// This is what lets a reporter be slow without blocking a test. Anything that

// takes time - a file write, an ADS call - is STARTED in one of the notification

// methods and ADVANCED here.
METHOD CyclicLogic
VAR
	i : DINT;
END_VAR
FOR i := 0 TO TO_DINT(_Count) - 1 DO
	_Reporters[i].CyclicLogic();
END_FOR
END_METHOD

// Never silent, and never reported as a test failure.

//

// Reaching here with nothing attached IS silent, and there is nothing this object

// can do about it. That is what ReporterCount exists for: assert it in CI.
METHOD FrameworkError
VAR_INPUT
	Source	: T_MaxString;
	Message : T_MaxString;
END_VAR

VAR
	i : DINT;
END_VAR
IF _IsSuspended THEN
	RETURN;
END_IF

FOR i := 0 TO TO_DINT(_Count) - 1 DO
	_Reporters[i].FrameworkError(Source := Source, Message := Message);
END_FOR
END_METHOD

// FALSE while ANY attached sink still has work in flight.

//

// CI must wait for this as well as IsComplete. A run finishing and its result

// document reaching disk are different events, and copying between them yields a

// truncated artifact - which reads as a broken pipeline rather than a finished

// run.

//

// TRUE with nothing attached: no sink, no pending work.
PROPERTY IsIdle : BOOL
GET
VAR
	i : DINT;
END_VAR
IsIdle := TRUE;
FOR i := 0 TO TO_DINT(_Count) - 1 DO
	IF NOT _Reporters[i].IsIdle THEN
		IsIdle := FALSE;
		RETURN;
	END_IF
END_FOR
END_GET
END_PROPERTY

// Notify sinks again. Nothing that happened while suspended is replayed - it was

// deliberately not recorded.
METHOD Resume
_IsSuspended := FALSE;
END_METHOD

METHOD RunFinished
VAR_INPUT
	Status	   : I_TestRunStatus;
	TargetInfo : T_MaxString;
END_VAR

VAR
	i : DINT;
END_VAR
IF _IsSuspended THEN
	RETURN;
END_IF

FOR i := 0 TO TO_DINT(_Count) - 1 DO
	_Reporters[i].RunFinished(Status := Status, TargetInfo := TargetInfo);
END_FOR
END_METHOD

METHOD RunStarted
VAR_INPUT
	Label	   : T_MaxString;
	TargetInfo : T_MaxString;
END_VAR

VAR
	i : DINT;
END_VAR
IF _IsSuspended THEN
	RETURN;
END_IF

FOR i := 0 TO TO_DINT(_Count) - 1 DO
	_Reporters[i].RunStarted(Label := Label, TargetInfo := TargetInfo);
END_FOR
END_METHOD

METHOD SuiteFinished
VAR_INPUT
	Status : I_TestRunStatus;
END_VAR

VAR
	i : DINT;
END_VAR
IF _IsSuspended THEN
	RETURN;
END_IF

FOR i := 0 TO TO_DINT(_Count) - 1 DO
	_Reporters[i].SuiteFinished(Status);
END_FOR
END_METHOD

// Stop notifying sinks. Used for an individual re-run, which must not pollute the

// CI artifact with duplicate entries.

//

// Work already in flight is unaffected - CyclicLogic keeps running - so a document

// being written when this is called still lands.
METHOD Suspend
_IsSuspended := TRUE;
END_METHOD

METHOD TestFinished
VAR_INPUT
	SuiteLabel	  : T_MaxString;
	TestLabel	  : T_MaxString;
	Location	  : T_MaxString;
	Status		  : E_TestStatus;
	Kind		  : E_FailureKind;
	Summary		  : T_MaxString;
	ElapsedTime	  : LREAL;
	ElapsedCycles : UDINT;
	Assertions	  : UDINT;
END_VAR

VAR
	i : DINT;
END_VAR
IF _IsSuspended THEN
	RETURN;
END_IF

FOR i := 0 TO TO_DINT(_Count) - 1 DO
	_Reporters[i].TestFinished(SuiteLabel	 := SuiteLabel,
							   TestLabel	 := TestLabel,
							   Location		 := Location,
							   Status		 := Status,
							   Kind			 := Kind,
							   Summary		 := Summary,
							   ElapsedTime	 := ElapsedTime,
							   ElapsedCycles := ElapsedCycles,
							   Assertions	 := Assertions);
END_FOR
END_METHOD

// Only the sinks that asked for checks. A reporter that does not implement

// I_TestDetailSink is skipped without a query and without an empty method body.
METHOD TestStarted
VAR_INPUT
	SuiteLabel : T_MaxString;
	TestLabel  : T_MaxString;
	Location   : T_MaxString;
END_VAR

VAR
	i : DINT;
END_VAR
IF _IsSuspended THEN
	RETURN;
END_IF

FOR i := 0 TO TO_DINT(_Count) - 1 DO
	IF _DetailSinks[i] <> 0 THEN
		_DetailSinks[i].TestStarted(SuiteLabel := SuiteLabel, TestLabel := TestLabel, Location := Location);
	END_IF
END_FOR
END_METHOD

END_FUNCTION_BLOCK

// ---- POUs/TestArbiter.TcPOU
// Which test runs next, and when there are no more.

//

// Separated from the runner because it is the ordering POLICY and the runner is

// the test LIFECYCLE - two different reasons to change. Everything a sequencer

// parks for later lands here and nowhere else: stop on first failing test, retry,

// preconditions. Today it walks the set in registration order, and that is all it

// should do.

//

// Not generic, and holds nothing generic. It reaches the registered set through

// I_TestRoster, which is read-only: an object that decides what runs next has no

// business registering a test or clearing a verdict.
FUNCTION_BLOCK TestArbiter
VAR
	_Roster : I_TestRoster;

	// The active test. A null Test member means none - there is no sentinel index.
	_Current : ST_TestSlot;
	_Count	 : DINT;

	// Where the NEXT Advance will look. Not the active index: that lives on

	// _Current, which is the only place it is meaningful.
	_Next : DINT;

	// Never written. Assigned to _Current to clear it, so "nothing active" is one

	// well-defined value rather than six field assignments to keep in step.
	_EmptySlot : ST_TestSlot;
END_VAR

(*
	No cyclic body. Advance is called by the suite when the active test finishes,
	not every scan.
*)

// Stop the pass where it is. Called when Enable drops: the active test, and any

// setup or teardown in flight, are cancelled by the runner and the pass does not

// resume.

//

// The remaining tests are NOT visited. A run that was abandoned mid-way has not

// been run, and reporting the rest as anything - passed, failed, skipped - would

// be inventing a result.
METHOD Abandon
_Current := _EmptySlot;
_Next	 := _Count;
END_METHOD

// Move to the next test. Returns TRUE when there is one, FALSE when the pass is

// over.

//

// The return value is the whole "are we finished" mechanism, so a caller cannot

// reach a test without first having been told there is one.
METHOD Advance : BOOL
Advance	 := FALSE;
_Current := _EmptySlot;
IF (_Roster = 0) OR (_Next >= _Count) THEN
	_Next := _Count;
	RETURN;
END_IF

_Current := _Roster.Slot(_Next);
_Next	 := _Next + 1;

// A slot inside the registered range always carries a test. If one does not, the

// registry and the count disagree, and running nothing is safer than dereferencing

// a null.
Advance := (_Current.Test <> 0);
END_METHOD

// Point the arbiter at the registered set. Called once by the suite at

// composition, before any run.

//

// An interface, not the registry itself: TestRegistry is generic and cannot be

// held by its concrete type here. That constraint turned out to be the thing that

// is what makes that workable - an interface reference carries no

// generic argument, so the arbiter can hold the set AND stay non-generic.
METHOD Attach
VAR_INPUT
	Roster : I_TestRoster;
END_VAR
_Roster := Roster;
END_METHOD

// Start a pass over the registered set, in registration order.

//

// Also what a re-run calls: a re-run re-executes the registered set from the

// start, so there is no separate restart path to keep in step with this one.

//

// The count is read here, once, rather than per Advance. Registration is closed by

// the time a run starts, so it cannot change underneath the pass.
METHOD Begin
_Current := _EmptySlot;
_Next	 := 0;
IF _Roster = 0 THEN
	// Nothing attached. An empty pass rather than a fault: IsExhausted goes TRUE

	// immediately and the suite completes instead of waiting for a test that will
	// never come.
	_Count := 0;
	RETURN;
END_IF

_Count := TO_DINT(_Roster.Count);
END_METHOD

// The active test, with its label, its index and its resolved hooks. Its Test

// member is NULL when nothing is active, which is the question callers ask.

//

// "None" is a null reference, not a sentinel

// index. The index is still here - a slot carries its own position, so the runner

// can reach the matching journal - but it is carried BY the thing that is null

// when there is nothing, rather than standing in for it.
PROPERTY Current : ST_TestSlot
GET
Current := _Current;
END_GET
END_PROPERTY

// TRUE while a test is active.

//

// Letting index 0 double as "no active test" is the trap here, and the note

// why that could not work is what CHAR_SerialExecution pins. Here there is no

// index to misread: the question is whether a reference is null.
PROPERTY HasCurrent : BOOL
GET
HasCurrent := (_Current.Test <> 0);
END_GET
END_PROPERTY

// Every registered test has been visited, or the pass was abandoned. What the

// suite reads to decide the run is over.

//

// Both conditions are required. After the last test is selected the pass has

// nothing left to give out, but that test is still running - reporting the suite

// complete there would cut it off.

//

// TRUE immediately for a pass over an empty set: a suite with nothing registered

// is complete, not stuck, or any sequencer aggregating it waits forever.
PROPERTY IsExhausted : BOOL
GET
IsExhausted := (_Next >= _Count) AND (_Current.Test = 0);
END_GET
END_PROPERTY

END_FUNCTION_BLOCK

// ---- POUs/TestDeadline.TcPOU
// Bounds one phase that is not the test body: setup, or teardown.

//

// The body's deadline stays in TestJournal, which already counts that phase's

// scans and already owns the verdict an expiry produces. This object exists for

// the two phases nothing else is watching.

//

// Teardown is the reason it exists at all. TestJournal.Tick returns immediately

// once the verdict is terminal, and teardown runs after the verdict by

// definition - so before this, teardown had no deadline of any kind. On a rig

// that means an axis left powered.

//

// Self-contained: its own clock and its own scan count, because setup runs before

// the body has a first cycle and teardown runs after the journal has stopped.

// Neither span is one the journal is measuring.
FUNCTION_BLOCK TestDeadline
VAR
	_Phase		   : T_MaxString;
	_Budget		   : ST_TestBudget;
	_ElapsedCycles : UDINT;
	_Stopwatch	   : TestStopwatch;
	_IsArmed	   : BOOL;
	_Diagnostic	   : T_MaxString;
END_VAR

(*
	No cyclic body. Tick is called by the runner while the phase is in progress,
	and only then.
*)

// Start bounding a phase. Restarts the clock and the scan count.

//

// The budget passed here is the RESOLVED one - the test's own, or the suite

// default it inherited. The IsSet flags have already done their work by this

// point and are not read.
METHOD Arm
VAR_INPUT
	// 'setup' or 'teardown'. Appears in the diagnostic, so a reader can tell which

	// phase hung without opening the test.
	Phase  : T_MaxString;
	Budget : ST_TestBudget;
END_VAR
_Phase		   := Phase;
_Budget		   := Budget;
_ElapsedCycles := 0;
_Diagnostic	   := '';
_IsArmed	   := TRUE;
_Stopwatch.Start();
END_METHOD

// Why it expired, in the shared wording. Empty until it does.
PROPERTY Diagnostic : T_MaxString
GET
Diagnostic := _Diagnostic;
END_GET
END_PROPERTY

// The phase finished on its own. Stops the clock and leaves any diagnostic

// already composed intact.
METHOD Disarm
_IsArmed := FALSE;
_Stopwatch.Stop();
END_METHOD

// Scans this phase has consumed.
PROPERTY ElapsedCycles : UDINT
GET
ElapsedCycles := _ElapsedCycles;
END_GET
END_PROPERTY

PROPERTY IsArmed : BOOL
GET
IsArmed := _IsArmed;
END_GET
END_PROPERTY

// Advance one scan. Returns TRUE on the scan the deadline expires, and FALSE

// every scan after that - the caller acts once.

//

// Called AFTER the phase has run, so a budget of one allows one execution. This

// matches TestJournal.Tick deliberately: two deadline mechanisms that counted

// differently would be a trap.
METHOD Tick : BOOL
Tick := FALSE;
IF NOT _IsArmed THEN
	RETURN;
END_IF

_ElapsedCycles := _ElapsedCycles + 1;
IF (_Budget.Cycles > 0) AND (_ElapsedCycles >= _Budget.Cycles) THEN
	_Diagnostic := TestTimeoutDiagnostic(Phase	  := _Phase,
										 Cycles	  := _Budget.Cycles,
										 Timeout  := _Budget.Timeout,
										 ByCycles := TRUE);

	THIS^.Disarm();
	Tick := TRUE;
	RETURN;
END_IF

IF (_Budget.Timeout > T#0S) AND (_Stopwatch.Elapsed >= (TO_LREAL(TIME_TO_UDINT(_Budget.Timeout)) / 1000.0)) THEN
	_Diagnostic := TestTimeoutDiagnostic(Phase	  := _Phase,
										 Cycles	  := _Budget.Cycles,
										 Timeout  := _Budget.Timeout,
										 ByCycles := FALSE);

	THIS^.Disarm();
	Tick := TRUE;
END_IF
END_METHOD

END_FUNCTION_BLOCK

// ---- POUs/TestEventReporter.TcPOU
// Raises TwinCAT 3 EventLogger events for test results.

//

// The sink for anything an operator or an HMI will see: structured, timestamped,

// localizable, and filterable by event class and ID - which ADSLOGSTR output is

// not. TestLogReporter remains the sink to reach for when no project setup is

// wanted.

//

// REQUIRES the TestHarnessEvents event class in the System Type System. TwinCAT

// generates TC_Events.TestHarnessEvents from it, and every event raised below is a

// member of that.

//

// Naming the generated members rather than a GUID is deliberate: if the class is

// not registered the symbol does not resolve and this FAILS TO COMPILE, which is a

// far better failure than raising events the logger has no name for.

//

// Severity comes from the class definition too, so it is declared once - one event

// ID per outcome, each carrying its own severity.

//

// It implements I_TestReporter and NOT I_TestDetailSink. An operator-facing log

// wants verdicts; an event per individual check would bury them.

//

// Severity is not decoration. A FAILURE is Error - the code was shown to be wrong.

// An ERROR is Warning - the test could not run, so nothing was shown about the

// code at all. A build should react differently to each, and so should whoever is

// looking at the Logged Events window.
FUNCTION_BLOCK TestEventReporter IMPLEMENTS I_TestReporter
VAR
	_Message	   : FB_TcMessage;
	_IncludePasses : BOOL;
	_EventsSent	   : UDINT;
	_FailedSends   : UDINT;
	_LastError	   : HRESULT;
END_VAR

(*
	No cyclic body. Everything this sink does happens inside the notification that
	prompted it.
*)

// Nothing to advance. Send hands the message to the EventLogger and returns; the

// logger owns what happens next.
METHOD CyclicLogic
(*
	Deliberately empty. This sink starts no work it has to finish, which is also
	why IsIdle is always TRUE.
*)
END_METHOD

// The one place an event is raised. Private, so the class, the severity mapping

// and the argument handling cannot drift between call sites.
METHOD Emit
VAR_INPUT
	// A member of TC_Events.TestHarnessEvents. Carries the class GUID, the ID and

	// the severity, all three declared once in the .tmc.
	EventEntry : TcEventEntry;
	Line	   : T_MaxString;
END_VAR

VAR
	Arguments : I_TcArguments;
	Result	  : HRESULT;
END_VAR
// CreateEx, not Create: it takes the whole definition, so the class, the ID and

// the severity all come from the .tmc and none of them is restated here.

//

// ipSourceInfo 0 means "generate it", which yields the symbol path of this

// instance - the reason a raised event names the test that raised it without
// being told.
Result := _Message.CreateEx(stEventEntry := EventEntry, ipSourceInfo := 0);
IF Result < 0 THEN
	_LastError	 := Result;
	_FailedSends := _FailedSends + 1;
	RETURN;
END_IF

// ipArguments is a PROPERTY returning an interface. TwinCAT will not take a member

// off the result of a call, so it goes into a variable first.
Arguments := _Message.ipArguments;
IF Arguments <> 0 THEN
	// Cleared every time: the instance is reused, and arguments left over from the
	// previous event would be appended to this one.
	Arguments.Clear();
	Arguments.AddString(Line);
END_IF

// 0 means "use the current timestamp".
Result := _Message.Send(0);
IF Result < 0 THEN
	_LastError	 := Result;
	_FailedSends := _FailedSends + 1;
	RETURN;
END_IF

_EventsSent := _EventsSent + 1;

// Release the instance the logger created. Without it, a long run leaks one per

// event - which would show up as memory growth rather than as anything obviously

// wrong with the test results.
_Message.Release();
END_METHOD

// Events accepted by the logger. Assert it in CI if events are the artifact.
PROPERTY EventsSent : UDINT
GET
EventsSent := _EventsSent;
END_GET
END_PROPERTY

// Create or Send returned a failing HRESULT.

//

// Counted rather than swallowed. A sink that cannot deliver and cannot say so is

// indistinguishable from a run that never happened.
PROPERTY FailedSends : UDINT
GET
FailedSends := _FailedSends;
END_GET
END_PROPERTY

METHOD FrameworkError
VAR_INPUT
	Source	: T_MaxString;
	Message : T_MaxString;
END_VAR
// Never silent, never suppressed by verbosity, and never reported as a test

// failure. This is the framework saying it could not do something.

//

// One ID for every framework error. The alternative was an event class growing a

// member for each new kind, which puts the class and this file permanently in step
// with each other.
THIS^.Emit(TC_Events.TestHarnessEvents.RegistrationRejected, CONCAT(CONCAT(Source, ': '), Message));
END_METHOD

// Always TRUE. Send hands the message over and returns; this sink never holds a

// run open waiting for the logger.
PROPERTY IsIdle : BOOL
GET
IsIdle := TRUE;
END_GET
END_PROPERTY

// The most recent failing HRESULT, or zero. 16#0 means nothing has gone wrong.
PROPERTY LastError : HRESULT
GET
LastError := _LastError;
END_GET
END_PROPERTY

METHOD RunFinished
VAR_INPUT
	Status	   : I_TestRunStatus;
	TargetInfo : T_MaxString;
END_VAR

VAR
	Line	: T_MaxString;
	Outcome : E_RunOutcome;
END_VAR
IF Status = 0 THEN
	RETURN;
END_IF

// TargetInfo identifies where the run happened. Without it a matrix run across

// several targets produces events that cannot be told apart.
Line := CONCAT(CONCAT(THIS^.Tally(Status), '  on '), TargetInfo);
// Read into a variable, as SuiteFinished does: TwinCAT will not take a CASE
// selector off a property call.
Outcome := Status.Outcome;
// The same four outcomes as the suite, each with its own event. RunSkipped and
// RunErrored were added to the class for this: a skipped run is not red, and an
// errored one showed nothing about the code, so neither is a RunFailed.
CASE Outcome OF
	E_RunOutcome.Passed:
		THIS^.Emit(TC_Events.TestHarnessEvents.RunPassed, Line);
	E_RunOutcome.Skipped:
		THIS^.Emit(TC_Events.TestHarnessEvents.RunSkipped, Line);
	E_RunOutcome.Errored:
		THIS^.Emit(TC_Events.TestHarnessEvents.RunErrored, Line);
ELSE
	THIS^.Emit(TC_Events.TestHarnessEvents.RunFailed, Line);
END_CASE
END_METHOD

// Deliberately raises nothing.

//

// A banner is a LOG device: it exists because log lines are an undifferentiated

// stream that a reader scrolls through. Events are already discrete, timestamped

// and filterable by class and ID, so bracketing them would add noise to a view

// that does not need it.
METHOD RunStarted
VAR_INPUT
	Label	   : T_MaxString;
	TargetInfo : T_MaxString;
END_VAR
(*
	Nothing. See the declaration.
*)
END_METHOD

// Whether passing tests raise an event of their own. Skipped tests do not: the

// event class has no per-test skipped event, so a skip is carried by the suite's

// SuiteSkipped event until the class gains one.

//

// Off by default. Eighty Info events bury the two Errors, and the counts are

// already available through I_TestRunStatus. The Verbose severity exists for this

// and is filtered out of most views anyway - but not raising them at all is

// cheaper still.
METHOD SetVerbosity
VAR_INPUT
	IncludePasses : BOOL;
END_VAR
_IncludePasses := IncludePasses;
END_METHOD

METHOD SuiteFinished
VAR_INPUT
	Status : I_TestRunStatus;
END_VAR

VAR
	Line	: T_MaxString;
	Outcome : E_RunOutcome;
END_VAR
IF Status = 0 THEN
	RETURN;
END_IF

Line := CONCAT(CONCAT(Status.Label, ': '), THIS^.Tally(Status));

// Read into a variable: a property call is a call, and TwinCAT will not take a

// CASE selector off one any more than it will take a member.
Outcome := Status.Outcome;
// A distinct event ID per outcome, so a filtered view can show suite results

// without showing every individual failure.
CASE Outcome OF
	E_RunOutcome.Passed:
		THIS^.Emit(TC_Events.TestHarnessEvents.SuitePassed, Line);

	E_RunOutcome.Skipped:
		THIS^.Emit(TC_Events.TestHarnessEvents.SuiteSkipped, Line);

	E_RunOutcome.Errored:
		THIS^.Emit(TC_Events.TestHarnessEvents.SuiteErrored, Line);

ELSE
	THIS^.Emit(TC_Events.TestHarnessEvents.SuiteFailed, Line);
END_CASE
END_METHOD

// The counts as one readable phrase. Shared by the suite and run events so the two

// cannot drift apart.
METHOD Tally : T_MaxString
VAR_INPUT
	Status : I_TestRunStatus;
END_VAR
IF Status = 0 THEN
	RETURN;
END_IF

Tally := CONCAT(UDINT_TO_STRING(Status.PassedCount), ' passed');
Tally := CONCAT(Tally, CONCAT(', ', UDINT_TO_STRING(Status.FailedCount)));
Tally := CONCAT(Tally, ' failed');
Tally := CONCAT(Tally, CONCAT(', ', UDINT_TO_STRING(Status.ErrorCount)));
Tally := CONCAT(Tally, ' errored');
Tally := CONCAT(Tally, CONCAT(', ', UDINT_TO_STRING(Status.SkippedCount)));
Tally := CONCAT(Tally, ' skipped, of ');
Tally := CONCAT(Tally, UDINT_TO_STRING(Status.TestCount));
END_METHOD

METHOD TestFinished
VAR_INPUT
	SuiteLabel	  : T_MaxString;
	TestLabel	  : T_MaxString;
	Location	  : T_MaxString;
	Status		  : E_TestStatus;
	Kind		  : E_FailureKind;
	Summary		  : T_MaxString;
	ElapsedTime	  : LREAL;
	ElapsedCycles : UDINT;
	Assertions	  : UDINT;
END_VAR

VAR
	Line : T_MaxString;
END_VAR
Line := CONCAT(CONCAT(SuiteLabel, ' / '), TestLabel);
CASE Status OF
	E_TestStatus.Failed:
		THIS^.Emit(TC_Events.TestHarnessEvents.TestFailed, CONCAT(CONCAT(Line, ': '), Summary));

	E_TestStatus.Errored:
		// Warning, not Error. The code under test was never shown to be wrong, and a
		// build should react differently to the two.
		THIS^.Emit(TC_Events.TestHarnessEvents.TestErrored, CONCAT(CONCAT(Line, ': '), Summary));

ELSE
	// Passes only. The event class has no per-test skipped event, and TestPassed for
	// a skipped test would report work that never ran; the suite's SuiteSkipped
	// event carries the count instead.
	IF _IncludePasses AND (Status = E_TestStatus.Passed) THEN
		THIS^.Emit(TC_Events.TestHarnessEvents.TestPassed, Line);
	END_IF
END_CASE
END_METHOD

END_FUNCTION_BLOCK

// ---- POUs/TestJUnitReporter.TcPOU
// Writes the run as a JUnit XML document - the artifact CI actually consumes.

//

// Implements BOTH reporter faces. I_TestReporter for verdicts and totals,

// I_TestDetailSink for individual checks, because this is the sink that detail

// streaming was designed for: every failed check becomes its own element rather

// than text appended to a growing string.

//

// That is what sidesteps the 255-character ceiling. CONCAT cannot build a longer

// string than that, so a document assembled by concatenation would truncate.

// Assembled as a DOM, no single value ever needs to exceed 255 - the document

// grows by nodes, not by characters.

//

// A DOM rather than streamed text, for one reason above the others: ESCAPING. Test

// labels are author-written and the compared values come from the code under

// test - arbitrary bytes by design. A hand-rolled escape that is subtly wrong

// produces a corrupt document rather than a visible error, and works for a year

// first.

//

// THE WRITE IS ASYNCHRONOUS and driven from CyclicLogic. IsIdle is FALSE until the

// file lands.

//

// ONE RUN, ONE FILE. Nothing is written per suite: a partially written artifact

// read by CI is worse than a missing one, because it looks complete.
FUNCTION_BLOCK TestJUnitReporter IMPLEMENTS I_TestReporter, I_TestDetailSink
VAR
	_Parser	   : FB_XmlDomParser;
	_RootNode  : SXmlNode;
	_SuiteNode : SXmlNode;
	_CaseNode  : SXmlNode;

	// Node validity is tracked with flags rather than by inspecting SXmlNode. What

	// an unset one contains is not something to rely on.
	_HasDocument  : BOOL;
	_HasSuiteNode : BOOL;
	_HasCaseNode  : BOOL;
	_Path		  : T_MaxString;
	_IsSaving	  : BOOL;
	_PassedChecks : UDINT;
	_FailedChecks : UDINT;

	// Where a failed write is reported. Never this object's own fan-out - that

	// would call back into here.
	_Reporter		 : I_TestReporter;
	_FilesWritten	 : UDINT;
	_WriteFailures	 : UDINT;
	_FrameworkErrors : UDINT;
	_LastError		 : HRESULT;
END_VAR

(*
	No cyclic body. CyclicLogic is the cyclic entry point and is called by the
	fan-out, which is called by the suite.
*)

// Where a failed write is reported. Optional but strongly advised.

//

// Without it, the only evidence of a failed write is WriteFailures on this object.

// A sink that cannot write its file and cannot say so is silent about the one

// thing that matters.

//

// Deliberately not the fan-out this object is attached to: reporting a write

// failure back through the composite would call this object again.
METHOD AttachErrorSink
VAR_INPUT
	Reporter : I_TestReporter;
END_VAR
_Reporter := Reporter;
END_METHOD

// Start a fresh document. Called on the first result of a run, and again by

// ReRun - a re-run produces a fresh document rather than appending to the last.
METHOD BeginDocument
VAR
	DocumentNode : SXmlNode;
END_VAR
IF _HasDocument THEN
	RETURN;
END_IF

_Parser.NewDocument();

// GetDocumentNode is what an element attaches to. GetRootNode returns the first

// ELEMENT, which an empty document does not have.
DocumentNode := _Parser.GetDocumentNode();

// The JUnit root. Several suites can sit under it, which is what a sequencer

// produces.
_RootNode	  := _Parser.AppendNode(DocumentNode, 'testsuites');
_HasDocument  := TRUE;
_HasSuiteNode := FALSE;
_HasCaseNode  := FALSE;
END_METHOD

// Open a testsuite element the first time a result arrives for it.

//

// Attributes are filled in at SuiteFinished, when the counts are known - a

// testsuite element carries totals that do not exist while it is running.
METHOD BeginSuite
VAR_INPUT
	SuiteLabel : T_MaxString;
END_VAR
THIS^.BeginDocument();
IF _HasSuiteNode THEN
	RETURN;
END_IF

_SuiteNode	  := _Parser.AppendNode(_RootNode, 'testsuite');
_HasSuiteNode := TRUE;
_Parser.AppendAttribute(_SuiteNode, 'name', SuiteLabel);
END_METHOD

// EVERY failed check gets its own element - not just the first.

//

// This is what the streamed detail was for. The summary keeps only the first

// failure because 80 characters has room for one; the document has room for all of

// them, and each is a separate element rather than a growing string. That

// sidesteps the 255-character ceiling entirely: no single value here can exceed

// it, so nothing has to be truncated to fit.

//

// Expected and Actual go in their own attributes, in full, exactly as they arrived.
METHOD CheckFailed
VAR_INPUT
	StepLabel  : T_MaxString;
	Kind	   : E_FailureKind;
	Expected   : T_MaxString;
	Actual	   : T_MaxString;
	Diagnostic : T_MaxString;
	Message	   : T_MaxString;
END_VAR

VAR
	CheckNode : SXmlNode;
END_VAR
IF NOT _HasCaseNode THEN
	RETURN;
END_IF

_FailedChecks := _FailedChecks + 1;
CheckNode	  := _Parser.AppendNode(_CaseNode, 'check');
_Parser.AppendAttribute(CheckNode, 'step', StepLabel);
_Parser.AppendAttribute(CheckNode, 'expected', Expected);
_Parser.AppendAttribute(CheckNode, 'actual', Actual);
_Parser.AppendAttribute(CheckNode, 'diagnostic', Diagnostic);
_Parser.AppendAttribute(CheckNode, 'message', Message);
END_METHOD

// Counted, not written. A document listing every satisfied check would be

// enormous and would say nothing a reader wants.
METHOD CheckPassed
VAR_INPUT
	StepLabel : T_MaxString;
	Detail	  : T_MaxString;
END_VAR
_PassedChecks := _PassedChecks + 1;
END_METHOD

// Advances the file write. This is the sink the cyclic method exists for: a DOM

// save is asynchronous and cannot complete in the cycle that asked for it.

//

// SaveDocumentToFile clears the flag it was given when the write finishes, and its

// return value is meaningful on that one call - so the result is captured on the

// transition, not polled for afterwards.
METHOD CyclicLogic
VAR
	Finished : BOOL;
	Written	 : BOOL;
	Error	 : HRESULT;
END_VAR
IF NOT _IsSaving THEN
	RETURN;
END_IF

Written := _Parser.SaveDocumentToFile(sFile := _Path, bExec := _IsSaving, hrErrorCode => Error);

// The method resets _IsSaving when the asynchronous write ends.
Finished := NOT _IsSaving;
IF NOT Finished THEN
	RETURN;
END_IF

// The document has been written, so the next run starts a fresh one. Cleared here

// rather than when the write was requested, so nothing can replace the DOM while

// it is still being read.
_HasDocument := FALSE;
IF Written THEN
	_FilesWritten := _FilesWritten + 1;
	RETURN;
END_IF

// A write that failed is REPORTED, not discarded. Throwing away the FALSE and the

// HRESULT makes a bad path indistinguishable from a suite that never finished.
_WriteFailures := _WriteFailures + 1;
_LastError	   := Error;
IF _Reporter <> 0 THEN
	_Reporter.FrameworkError('TestJUnitReporter', CONCAT('the result document could not be written to ', _Path));
END_IF
END_METHOD

// Size of the document currently in DOM memory, in bytes.

//

// Exposed so a test can prove the document is not EMPTY. Nothing in the PLC reads

// the written file back, and a successful write of an empty document is

// indistinguishable from a successful write of a full one.
PROPERTY DocumentLength : UDINT
GET
DocumentLength := _Parser.GetDocumentLength();
END_GET
END_PROPERTY

// Documents successfully written. One per run.
PROPERTY FilesWritten : UDINT
GET
FilesWritten := _FilesWritten;
END_GET
END_PROPERTY

// Recorded in the document, so a run that could not be trusted says so in the

// artifact rather than only in a log nobody kept.

//

// Not a testcase: it is not a test, and counting it as one would corrupt the

// totals CI reads.
METHOD FrameworkError
VAR_INPUT
	Source	: T_MaxString;
	Message : T_MaxString;
END_VAR

VAR
	ErrorNode : SXmlNode;
END_VAR
THIS^.BeginDocument();
ErrorNode := _Parser.AppendNode(_RootNode, 'framework-error');
_Parser.AppendAttribute(ErrorNode, 'source', Source);
_Parser.AppendAttribute(ErrorNode, 'message', Message);
_FrameworkErrors := _FrameworkErrors + 1;
END_METHOD

PROPERTY FrameworkErrors : UDINT
GET
FrameworkErrors := _FrameworkErrors;
END_GET
END_PROPERTY

// FALSE while the document is being written.

//

// CI must wait for this as well as IsComplete. A run finishing and its file

// reaching disk are different events, and copying between them yields a truncated

// artifact - which reads as a broken pipeline rather than a finished run.
PROPERTY IsIdle : BOOL
GET
IsIdle := NOT _IsSaving;
END_GET
END_PROPERTY

// The failure kind as the string CI groups by. A CASE rather than a lookup table

// because there are six of them and a table would be one more thing to keep in

// step with the enum.
METHOD KindName : T_MaxString
VAR_INPUT
	Kind : E_FailureKind;
END_VAR
CASE Kind OF
	E_FailureKind.ValueMismatch:
		KindName := 'ValueMismatch';

	E_FailureKind.TypeMismatch:
		KindName := 'TypeMismatch';

	E_FailureKind.SizeMismatch:
		KindName := 'SizeMismatch';

	E_FailureKind.Timeout:
		KindName := 'Timeout';

	E_FailureKind.Environment:
		KindName := 'Environment';

ELSE
	KindName := 'None';
END_CASE
END_METHOD

// The HRESULT from the most recent failed write, or zero.
PROPERTY LastError : HRESULT
GET
LastError := _LastError;
END_GET
END_PROPERTY

// Every suite is done. Requests the write.

//

// The document is NOT written per suite. One run, one file - a partially written

// artifact read by CI is worse than a missing one, because it looks complete.
METHOD RunFinished
VAR_INPUT
	Status	   : I_TestRunStatus;
	TargetInfo : T_MaxString;
END_VAR
IF NOT _HasDocument THEN
	// No document was ever opened, which means RunStarted never arrived - this sink

	// was never part of a run. Writing now would invent an artifact for something

	// that did not happen.

	//

	// An EMPTY run is different and does produce a document, carrying tests="0".

	// That was the opposite of the behaviour before RunStarted existed, and the

	// change is deliberate: a missing file is ambiguous - a configuration problem

	// and a run with no tests look identical - while tests="0" says which. It is the
	// same reasoning as R3, one level up.
	RETURN;
END_IF

IF TargetInfo <> '' THEN
	// Which target produced this. Without it a matrix run yields documents that
	// cannot be told apart.
	_Parser.AppendAttribute(_RootNode, 'target', TargetInfo);
END_IF

IF _Path = '' THEN
	IF _Reporter <> 0 THEN
		_Reporter.FrameworkError('TestJUnitReporter', 'no result path was set - call SetPath at composition');
	END_IF

	_WriteFailures := _WriteFailures + 1;
	RETURN;
END_IF

// CyclicLogic drives it from here. IsIdle stays FALSE until it lands, and CI must

// wait for that as well as IsComplete: a run finishing and its document reaching

// disk are different events.

//

// _HasDocument stays TRUE until the write COMPLETES. Clearing it here would let a

// late notification call BeginDocument and wipe the DOM out from under the write

// in progress.
_IsSaving := TRUE;
END_METHOD

// Opens the document, at the point the run says it has begun rather than when the

// first result happens to arrive.
METHOD RunStarted
VAR_INPUT
	Label	   : T_MaxString;
	TargetInfo : T_MaxString;
END_VAR
THIS^.BeginDocument();
END_METHOD

// Absolute path of the result document. REQUIRED - there is no default.

//

// The boot folder is where this belongs on a target. On build 4026 the Windows

// location moved to ProgramData - the 4024 path under C:\TwinCAT is wrong and

// writes nowhere useful:

//

//   C:\ProgramData\Beckhoff\TwinCAT\3.1\Boot\TestResults.xml   Windows, 4026

//   /usr/local/etc/TwinCAT/3.1/Boot/TestResults.xml            TwinCAT/BSD

//

// Which is the reason there is no default: the right answer depends on the build

// and the platform, and a wrong one writes somewhere nobody looks.

//

// Deliberately not defaulted. A default that is wrong for the platform writes

// somewhere nobody looks, and a missing file is indistinguishable from a run that

// never finished.
METHOD SetPath
VAR_INPUT
	Path : T_MaxString;
END_VAR
_Path := Path;
END_METHOD

// Fills in the totals a testsuite element carries, now that they exist.
METHOD SuiteFinished
VAR_INPUT
	Status : I_TestRunStatus;
END_VAR

VAR
	// AppendAttribute takes its value as VAR_IN_OUT CONSTANT, which needs something

	// with an address. A literal has one; the result of a call does not, so

	// anything computed goes into a local first.
	TimeText : T_MaxString;
END_VAR
IF Status = 0 THEN
	RETURN;
END_IF

THIS^.BeginSuite(Status.Label);
_Parser.AppendAttributeAsUint(_SuiteNode, 'tests', Status.TestCount);
_Parser.AppendAttributeAsUint(_SuiteNode, 'failures', Status.FailedCount);
_Parser.AppendAttributeAsUint(_SuiteNode, 'errors', Status.ErrorCount);
_Parser.AppendAttributeAsUint(_SuiteNode, 'skipped', Status.SkippedCount);
TimeText := LREAL_TO_FMTSTR(Status.TotalDuration, 6, TRUE);
_Parser.AppendAttribute(_SuiteNode, 'time', TimeText);

// The next suite opens its own element. A sequencer driving several produces

// several, all under one testsuites root.
_HasSuiteNode := FALSE;
END_METHOD

// Closes the testcase element with its verdict.

//

// A testcase with no child element is a pass - that is JUnit's convention, not an

// omission. Failure, error and skipped are each a distinct child, because CI

// counts them separately and so should this.
METHOD TestFinished
VAR_INPUT
	SuiteLabel	  : T_MaxString;
	TestLabel	  : T_MaxString;
	Location	  : T_MaxString;
	Status		  : E_TestStatus;
	Kind		  : E_FailureKind;
	Summary		  : T_MaxString;
	ElapsedTime	  : LREAL;
	ElapsedCycles : UDINT;
	Assertions	  : UDINT;
END_VAR

VAR
	VerdictNode : SXmlNode;

	// AppendAttribute takes its value as VAR_IN_OUT CONSTANT, which needs something

	// with an address. A literal has one; the result of a call does not, so

	// anything computed goes into a local first.
	TimeText : T_MaxString;
	TypeText : T_MaxString;
END_VAR
IF NOT _HasCaseNode THEN
	// No TestStarted arrived - a skipped test never becomes active. Open the
	// element now so the result is not lost.
	THIS^.TestStarted(SuiteLabel := SuiteLabel, TestLabel := TestLabel, Location := Location);
END_IF

IF NOT _HasCaseNode THEN
	RETURN;
END_IF

TimeText := LREAL_TO_FMTSTR(ElapsedTime, 6, TRUE);
_Parser.AppendAttribute(_CaseNode, 'time', TimeText);
_Parser.AppendAttributeAsUint(_CaseNode, 'cycles', ElapsedCycles);
_Parser.AppendAttributeAsUint(_CaseNode, 'assertions', Assertions);

// The split, not just the total. A test reporting 12 assertions of which 3 failed

// is a different situation from one reporting 12 that all passed, and the summary

// only ever names the first failure.
_Parser.AppendAttributeAsUint(_CaseNode, 'checks-passed', _PassedChecks);
_Parser.AppendAttributeAsUint(_CaseNode, 'checks-failed', _FailedChecks);
CASE Status OF
	E_TestStatus.Failed:
		// AppendChild, not AppendNode: it sets the element's BODY as well as creating

		// it, and the body is what a CI UI shows when someone clicks a failed test. An

		// attribute-only failure displays the message and nothing else.

		//

		// cdata TRUE so the summary needs no escaping of its own - it may contain
		// compared values, which are arbitrary bytes by design.
		VerdictNode := _Parser.AppendChild(_CaseNode,
										   'failure',
										   Summary,
										   TRUE);

		// The KIND goes in type, which is what CI groups by. The original hardcoded

		// 'AssertionError' for everything and made the field useless.
		TypeText := THIS^.KindName(Kind);
		_Parser.AppendAttribute(VerdictNode, 'type', TypeText);
		_Parser.AppendAttribute(VerdictNode, 'message', Summary);

	E_TestStatus.Errored:
		// error, not failure. The code under test was never shown to be wrong, and CI
		// keeps the two apart.
		VerdictNode := _Parser.AppendChild(_CaseNode,
										   'error',
										   Summary,
										   TRUE);

		TypeText := THIS^.KindName(Kind);
		_Parser.AppendAttribute(VerdictNode, 'type', TypeText);
		_Parser.AppendAttribute(VerdictNode, 'message', Summary);

	E_TestStatus.Skipped:
		VerdictNode := _Parser.AppendNode(_CaseNode, 'skipped');
END_CASE

_HasCaseNode := FALSE;
END_METHOD

// A test became the active one. Opens its testcase element, so the checks that

// follow have somewhere to go.

//

// This is why I_TestDetailSink has a TestStarted at all: checks arrive before the

// test has a verdict, and a document builder needs to be told when to open an

// element.
METHOD TestStarted
VAR_INPUT
	SuiteLabel : T_MaxString;
	TestLabel  : T_MaxString;
	Location   : T_MaxString;
END_VAR
THIS^.BeginSuite(SuiteLabel);
_CaseNode	  := _Parser.AppendNode(_SuiteNode, 'testcase');
_HasCaseNode  := TRUE;
_FailedChecks := 0;
_PassedChecks := 0;
_Parser.AppendAttribute(_CaseNode, 'name', TestLabel);

// classname is where to LOOK when a test fails. Empty when the test does not

// implement I_TestLocation, which is the common case and not a problem.
_Parser.AppendAttribute(_CaseNode, 'classname', Location);
END_METHOD

// Writes that failed, or were asked for with no path. Never silent - each also

// raises a framework error through the attached sink.
PROPERTY WriteFailures : UDINT
GET
WriteFailures := _WriteFailures;
END_GET
END_PROPERTY

END_FUNCTION_BLOCK

// ---- POUs/TestSuite.TcPOU
// The composition root's handle on a set of tests, and the sequencer's handle on

// running them. Six interfaces, four audiences, one object.

//

// It is a FACADE and should stay one. Registration lives in TestRegistry,

// ordering in TestArbiter, the test lifecycle in TestRunner, the counts in

// TestRunTally, the sinks in TestReporterFanout. What is left here is the

// registration window, the per-scan order of operations, and naming a framework

// error - and if this object grows past that, something belongs in one of the

// five.

//

// One object doing all six jobs is most of why such a thing becomes

// being replaced.

//

// GENERIC only because it declares TestRegistry<Capacity> as a member and only a

// generic can forward the argument. Nothing here is sized by Capacity. Everything

// else it owns is plain, and reaches the registry through interfaces this object

// hands out.
FUNCTION_BLOCK TestSuite
VAR_GENERIC CONSTANT
	Capacity : UDINT := TestHarnessParameter.Capacity;
END_VAR IMPLEMENTS I_TestRegistration, I_TestDefaults, I_TestConfiguration, I_TestSuite, I_TestReRun
VAR
	_Registry  : TestRegistry<Capacity>;
	_Arbiter   : TestArbiter;
	_Runner	   : TestRunner;
	_Tally	   : TestRunTally;
	_Reporters : TestReporterFanout;

	// ONE per suite, not one per test. Only one test runs at a time, so the handle

	// is retargeted to whichever journal is active rather than allocated per slot.

	// At capacity 50 that is the difference between one copy of the assertion

	// machinery and fifty.
	_Verdict   : TestVerdict;
	_Label	   : T_MaxString;
	_Defaults  : ST_TestBudgets;
	_IsRunning : BOOL;
	_IsWired   : BOOL;

	// An individual re-run is in progress: one test, reported nowhere and counted

	// nowhere. The arbiter is not involved and the tally is not touched.
	_IsSingle : BOOL;

	// Skip has settled the counts but not yet told the sinks. They are told when

	// the run first drives this suite - after RunStarted, in its place in the

	// sequence. Skip is only allowed before that, when a sink may not even be

	// attached yet.
	_IsSkipPending : BOOL;

	// The suite was skipped, for good. Skip is part of composition and a re-run does

	// not recompose, so ReRun reads this rather than running what was ruled out.
	_IsSkipped : BOOL;

	// Framework errors raised BEFORE the run started - a rejected registration, an

	// unnamed suite. Tally.Begin clears its counts, so these are held and re-applied

	// once the run exists. Without that, a test that failed to register would leave

	// the run green, which is the exact regression hazard the reporting exists for.
	_PendingErrors : UDINT;

	// The journal of the test that just finished, held so PublishTest can read it

	// after the runner has unloaded.
	_LastJournal	: REFERENCE TO TestJournal;
	_ActiveLocation : T_MaxString;
END_VAR

(*
	No cyclic body, deliberately. This object is reached through its interfaces -
	Register, Run, Skip - and a sequencer holding I_TestSuite has no way to call the
	function block itself. Wiring that depended on this running would silently never
	happen.

	EnsureWired is called from every entry point instead.
*)

METHOD AddReporter : BOOL
VAR_INPUT
	Reporter : I_TestReporter;
END_VAR
AddReporter := _Reporters.Attach(Reporter);
END_METHOD

// Hand the five collaborators to each other. Once, on first use.

//

// Not FB_init: the members are not all constructed when it runs. Not the cyclic

// body: this object is driven through its interfaces and the function block itself

// may never be called.
METHOD EnsureWired
IF _IsWired THEN
	RETURN;
END_IF

_IsWired := TRUE;
_Verdict.AttachDetailSink(_Reporters);
_Runner.Attach(Roster := _Registry, Verdict := _Verdict);
_Arbiter.Attach(_Registry);
END_METHOD

PROPERTY ErrorCount : UDINT
GET
ErrorCount := _Tally.ErrorCount;
END_GET
END_PROPERTY

PROPERTY FailedCount : UDINT
GET
FailedCount := _Tally.FailedCount;
END_GET
END_PROPERTY

// The pass is over, cleanly or by abandonment. Settles the aggregate and tells

// the sinks once.
METHOD FinishRun
IF NOT _IsRunning THEN
	RETURN;
END_IF

_IsRunning := FALSE;
_Tally.Finish();
_Reporters.SuiteFinished(THIS^);
END_METHOD

PROPERTY IsComplete : BOOL
GET
IsComplete := _Tally.IsComplete;
END_GET
END_PROPERTY

PROPERTY IsOpen : BOOL
GET
IsOpen := _Registry.IsOpen;
END_GET
END_PROPERTY

PROPERTY Label : T_MaxString
GET
Label := _Label;
END_GET
END_PROPERTY

PROPERTY Outcome : E_RunOutcome
GET
Outcome := _Tally.Outcome;
END_GET
END_PROPERTY

PROPERTY PassedCount : UDINT
GET
PassedCount := _Tally.PassedCount;
END_GET
END_PROPERTY

// One test reached a terminal state. Fold it into the totals and tell the sinks.
METHOD PublishTest
VAR
	Journal : REFERENCE TO TestJournal;
END_VAR
IF _IsSingle THEN
	// Records nothing. The verdict is visible in the journal for whoever is at the
	// keyboard; it does not reach the counts or the sinks.
	RETURN;
END_IF

Journal REF= _LastJournal;
IF NOT __ISVALIDREF(Journal) THEN
	RETURN;
END_IF

_Tally.Record(Verdict := Journal.Status, ElapsedTime := Journal.ElapsedTime);
_Reporters.TestFinished(SuiteLabel	  := _Label,
						TestLabel	  := Journal.Label,
						Location	  := Journal.Location,
						Status		  := Journal.Status,
						Kind		  := Journal.Kind,
						Summary		  := Journal.Summary,
						ElapsedTime	  := Journal.ElapsedTime,
						ElapsedCycles := Journal.ElapsedCycles,
						Assertions	  := Journal.AssertionCount);
END_METHOD

// One place framework errors are named, so every one of them carries this suite's

// label as its source.
METHOD RaiseFrameworkError
VAR_INPUT
	Message : T_MaxString;
END_VAR
IF _IsSingle THEN
	// An individual re-run is a debugging session, not a result. Its problems are
	// visible at the keyboard and must not turn a CI run red.
	RETURN;
END_IF

IF _IsRunning THEN
	_Tally.RecordFrameworkError();
ELSE
	// Held until there is a run to attribute it to.
	_PendingErrors := _PendingErrors + 1;
END_IF

_Reporters.FrameworkError(Source := _Label, Message := Message);
END_METHOD

METHOD Register : BOOL
VAR_INPUT
	Test	: I_Test;
	Label	: T_MaxString;
	Budgets : ST_TestBudgets;
END_VAR

VAR
	Fault : E_RegistrationFault;
END_VAR
THIS^.EnsureWired();
Fault	 := _Registry.TryClaim(Test := Test, Label := Label, Budgets := Budgets);
Register := (Fault = E_RegistrationFault.None);
IF Register THEN
	RETURN;
END_IF

// Never silent. A test that failed to register would otherwise vanish from the

// results and CI would see fewer passes rather than a failure - precisely the

// regression hazard RegisteredCount exists to catch.
CASE Fault OF
	E_RegistrationFault.Full:
		THIS^.RaiseFrameworkError(CONCAT('suite is full, rejected: ', Label));

	E_RegistrationFault.DuplicateLabel:
		THIS^.RaiseFrameworkError(CONCAT('label already registered: ', Label));

	E_RegistrationFault.EmptyLabel:
		THIS^.RaiseFrameworkError('a test was offered with no label');

	E_RegistrationFault.NoTest:
		THIS^.RaiseFrameworkError(CONCAT('no test supplied for label: ', Label));

	E_RegistrationFault.Closed:
		THIS^.RaiseFrameworkError(CONCAT('registration has closed, rejected: ', Label));
END_CASE
END_METHOD

PROPERTY RegisteredCount : UDINT
GET
RegisteredCount := _Registry.Count;
END_GET
END_PROPERTY

PROPERTY ReporterCount : UDINT
GET
ReporterCount := _Reporters.Count;
END_GET
END_PROPERTY

METHOD ReRun
IF _IsRunning THEN
	THIS^.RaiseFrameworkError('ReRun called while a run is in progress');
	RETURN;
END_IF

// A skipped suite stays skipped. A re-run "re-executes what was composed; it does
// not recompose it" (TestRun.ReRun), and a skip is part of what was composed - it
// is usually there because running these tests here would be wrong. Its verdicts
// and counts still stand, so nothing is reset; the suite is only announced again,
// when the run reaches it, so the fresh document still lists its tests.
IF _IsSkipped THEN
	_IsSkipPending := TRUE;
	RETURN;
END_IF

// The registered set is not redefined, only re-executed. The window stays shut.
_Registry.ResetAll();
THIS^.StartRun();
END_METHOD

METHOD ReRunSingle : BOOL
VAR_INPUT
	Label : T_MaxString;
END_VAR

VAR
	Index	: DINT;
	Slot	: ST_TestSlot;
	Journal : REFERENCE TO TestJournal;
END_VAR
THIS^.EnsureWired();
ReRunSingle := FALSE;
IF _IsRunning THEN
	// Not while the suite is running. Two tests writing the same fixtures is the
	// interference serial execution exists to prevent.
	RETURN;
END_IF

Index := _Registry.Lookup(Label);
IF Index < 0 THEN
	RETURN;
END_IF

Journal REF= _Registry.Journal(Index);
IF NOT __ISVALIDREF(Journal) THEN
	RETURN;
END_IF

Slot := _Registry.Slot(Index);

// Records nothing and saves nothing. Silencing the fan-out is the whole

// mechanism: a session at the keyboard cannot pollute the CI artifact with

// duplicate entries, and no condition has to be threaded through the runner.
_Reporters.Suspend();
Journal.Reset();
IF NOT _Runner.Load(Slot) THEN
	_Reporters.Resume();
	RETURN;
END_IF

_LastJournal REF= Journal;
_IsSingle	 := TRUE;
_IsRunning	 := TRUE;
ReRunSingle	 := TRUE;
END_METHOD

METHOD Run : BOOL
VAR_INPUT
	Enable : BOOL;
END_VAR

VAR
	Slot	: ST_TestSlot;
	Outcome : E_PhaseOutcome;
	i		: DINT;
	Journal : REFERENCE TO TestJournal;
	Location : T_MaxString;
END_VAR
THIS^.EnsureWired();

// Sinks advance whatever the suite is doing. A file write started at the end of

// the last run still has to finish, and a suite that has completed must keep

// pumping them or IsIdle never goes TRUE.
_Reporters.CyclicLogic();
Run := _Tally.IsComplete;
IF NOT Enable THEN
	IF _IsRunning THEN
		_Runner.Advance(Enable := FALSE);
		_Arbiter.Abandon();
		THIS^.FinishRun();
		Run := _Tally.IsComplete;
	END_IF

	RETURN;
END_IF

// A skipped suite is announced here, when the run reaches it. Skip already
// settled the counts, and nothing below would run a test.
//
// Each test first, by name, then the suite. The result document is read as
// cases, so a skipped test that is only a count is invisible to CI; and a
// document builder closes the suite element on SuiteFinished, so a case sent
// after it has nowhere to go. No TestStarted: a skipped test never became active,
// and the sinks already open the element themselves when one is missing.
IF _IsSkipPending THEN
	_IsSkipPending := FALSE;
	FOR i := 0 TO TO_DINT(_Registry.Count) - 1 DO
		Journal REF= _Registry.Journal(i);
		IF __ISVALIDREF(Journal) THEN
			// Label and location from the SLOT, the way TestRunner.Load takes them. A
			// journal only learns them in Begin, when its test becomes active - and a
			// skipped test never does, so its journal label is still empty.
			Slot	 := _Registry.Slot(i);
			Location := '';
			IF Slot.Location <> 0 THEN
				Location := Slot.Location.Path;
			END_IF

			_Reporters.TestFinished(SuiteLabel	  := _Label,
									TestLabel	  := Slot.Label,
									Location	  := Location,
									Status		  := Journal.Status,
									Kind		  := Journal.Kind,
									Summary		  := Journal.Summary,
									ElapsedTime	  := Journal.ElapsedTime,
									ElapsedCycles := Journal.ElapsedCycles,
									Assertions	  := Journal.AssertionCount);
		END_IF
	END_FOR

	_Reporters.SuiteFinished(THIS^);
	RETURN;
END_IF

IF _Registry.IsOpen THEN
	THIS^.StartRun();
END_IF

IF NOT _IsRunning THEN
	RETURN;
END_IF

Outcome := _Runner.Advance(Enable := TRUE);
CASE Outcome OF
	E_PhaseOutcome.Running:
		RETURN;

	E_PhaseOutcome.TeardownOverran:
		// The verdict stands - a passing test whose cleanup hung still proved the code

		// correct - but the run cannot be trusted, and on a rig this may mean an axis
		// left powered.
		THIS^.RaiseFrameworkError(CONCAT(CONCAT('teardown abandoned in ', _Runner.ActiveLabel), CONCAT(': ', _Runner.TeardownDiagnostic)));
		THIS^.PublishTest();

	E_PhaseOutcome.Finished:
		THIS^.PublishTest();
END_CASE

IF _IsSingle THEN
	// One test, done. Nothing was recorded and nothing was saved, so there is
	// nothing to settle - just put the sinks back.
	_IsSingle  := FALSE;
	_IsRunning := FALSE;
	_Reporters.Resume();
	Run := _Tally.IsComplete;
	RETURN;
END_IF

// Idle, or just finished one. Take the next.
IF _Arbiter.Advance() THEN
	Slot := _Arbiter.Current;
	IF NOT _Runner.Load(Slot) THEN
		// The arbiter offered something the runner would not take. Report it rather
		// than spinning on it.
		THIS^.RaiseFrameworkError(CONCAT('could not start test: ', Slot.Label));
		_Arbiter.Abandon();
		THIS^.FinishRun();
	ELSE
		// Held so PublishTest can read the record after the runner has unloaded.
		_LastJournal	REF= _Registry.Journal(Slot.Index);
		_ActiveLocation := '';
		IF __ISVALIDREF(_LastJournal) THEN
			_ActiveLocation := _LastJournal.Location;
		END_IF

		_Reporters.TestStarted(SuiteLabel := _Label, TestLabel := Slot.Label, Location := _ActiveLocation);
	END_IF
ELSIF _Arbiter.IsExhausted THEN
	THIS^.FinishRun();
END_IF

Run := _Tally.IsComplete;
END_METHOD

METHOD SetDefaults
VAR_INPUT
	Defaults : ST_TestBudgets;
END_VAR
// Stored, not applied. They reach the journals when the run starts, because a
// default may be set after some tests are already registered.
_Defaults := Defaults;
END_METHOD

METHOD SetLabel
VAR_INPUT
	Label : T_MaxString;
END_VAR
_Label := Label;
_Tally.SetLabel(Label);
END_METHOD

METHOD Skip
VAR
	i		: DINT;
	Journal : REFERENCE TO TestJournal;
END_VAR
THIS^.EnsureWired();
IF NOT _Registry.IsOpen THEN
	// Already enabled or already complete. Skipping now would rewrite results that
	// have been reported.
	THIS^.RaiseFrameworkError('Skip called after the suite was enabled');
	RETURN;
END_IF

// Closes the window. A skipped suite is complete, and registration does not

// reopen for a suite that has reached a terminal state.
_Registry.Close();
// The two checks StartRun makes before a pass, in the same order. A skip bypasses
// StartRun, and must not bypass these: a skipped suite still goes into the
// result document, and a wiring error is a wiring error whether or not the
// tests run. The label check comes first because, with no run yet, it adds to
// the pending errors re-applied below.
IF _Label = '' THEN
	THIS^.RaiseFrameworkError('suite was skipped with no label');
END_IF
_Tally.Begin(_Registry.Count);
// Tally.Begin cleared the counts. Re-apply anything raised before this point -
// a rejected registration above all - or it vanishes, and the run stays clear of
// red while a test is missing from it.
FOR i := 1 TO TO_DINT(_PendingErrors) DO
	_Tally.RecordFrameworkError();
END_FOR

FOR i := 0 TO TO_DINT(_Registry.Count) - 1 DO
	Journal REF= _Registry.Journal(i);
	IF __ISVALIDREF(Journal) THEN
		Journal.MarkSkipped();
		_Tally.Record(Verdict := E_TestStatus.Skipped, ElapsedTime := 0.0);
	END_IF
END_FOR

_Tally.Finish();
// Settled, but not announced. Skip runs before the suite is first enabled -
// before RunStarted, and often before any sink is attached - so an announcement
// made here reaches nothing, or arrives ahead of the run it belongs to. Run
// makes it when the run reaches this suite.
_IsSkipped	   := TRUE;
_IsSkipPending := TRUE;
END_METHOD

PROPERTY SkippedCount : UDINT
GET
SkippedCount := _Tally.SkippedCount;
END_GET
END_PROPERTY

// First enable, or a re-run. Closes the window, pushes the defaults into every

// journal, and starts the pass.
METHOD StartRun
VAR
	i : DINT;
END_VAR
_Registry.Close();
_Registry.ApplyDefaults(_Defaults);
// A re-run supersedes an announcement Skip left pending: the suite is about to
// report what it actually does.
_IsSkipPending := FALSE;
IF _Label = '' THEN
	// An unnamed suite produces an unnamed node in the result document, which no
	// CI system can group by.
	THIS^.RaiseFrameworkError('suite was enabled with no label');
END_IF

_Tally.Begin(_Registry.Count);
// Re-apply anything raised before the run existed, so a rejected registration

// still turns this run red.
FOR i := 1 TO TO_DINT(_PendingErrors) DO
	_Tally.RecordFrameworkError();
END_FOR

_Arbiter.Begin();
_IsRunning := TRUE;
END_METHOD

PROPERTY TestCount : UDINT
GET
TestCount := _Tally.TestCount;
END_GET
END_PROPERTY

PROPERTY TotalDuration : LREAL
GET
TotalDuration := _Tally.TotalDuration;
END_GET
END_PROPERTY

END_FUNCTION_BLOCK

// ---- POUs/TestRunner.TcPOU
// Drives ONE test through its three phases: setup, body, teardown.

//

// Separated from TestArbiter because that object decides WHICH test runs and this

// one decides WHAT HAPPENS to it - two different reasons to change. Separated from

// the suite because the suite is a facade and this is the only real state machine

// in the library.

//

// One instance per suite. Only one test runs at a time, which is the whole reason

// the verdict handle and the deadlines can be single copies rather than per slot.

//

// It holds no reporters. A teardown overrun is returned to the suite rather than

// reported here, because the suite is what owns the sinks - and keeping this

// object ignorant of them is what keeps it testable.
FUNCTION_BLOCK TestRunner
VAR
	_Roster : I_TestRoster;

	// A REFERENCE TO, not a copy. A function block held by value would be copied at

	// the call that supplied it, and the runner would retarget a copy nobody reads.
	_Verdict : REFERENCE TO TestVerdict;

	// The same object, as the interface a test body is handed. A REFERENCE TO does

	// not substitute for an interface at a call site, so it is held both ways.
	_Assertions : I_TestAssertions;
	_Slot		: ST_TestSlot;
	_Journal	: REFERENCE TO TestJournal;
	_Phase		: E_RunPhase;
	_Outcome	: E_PhaseOutcome;

	// Bounds setup and teardown. The BODY deadline lives in TestJournal, which

	// already counts that phase and already owns the verdict an expiry produces.
	_PhaseDeadline		: TestDeadline;
	_TeardownDiagnostic : T_MaxString;

	// The label of the test most recently loaded. NOT cleared by Unload.

	//

	// The suite reports a teardown overrun AFTER the runner has unloaded, so

	// reading the label off the slot at that point yields an empty string and the

	// framework error names no test at all. The diagnostic already survived Unload

	// for the same reason; the label has to as well.
	_LastLabel : T_MaxString;

	// Never written. Assigned to clear, so "nothing loaded" is one well-defined

	// value rather than six field assignments to keep in step.
	_EmptySlot : ST_TestSlot;
END_VAR

(*
	No cyclic body. Advance is called by the suite while a test is loaded, and only
	then.
*)

// Enable dropped. Give the phase in flight one final call so it can return its

// own state to its starting condition, then stop.

//

// The return value of that call is ignored. A test abandoned because it hung will

// not answer it either, and waiting for TRUE would reproduce the stall the whole

// design removes.

//

// Teardown is NOT run. Abandonment is the suite being switched off, not a test

// finishing, and calling cleanup on a half-torn-down rig is its own hazard.
METHOD Abandon
CASE _Phase OF
	E_RunPhase.Setup:
		_Slot.Setup.Setup(Enable := FALSE, Test := _Assertions);

	E_RunPhase.Body:
		_Slot.Test.Run(Enable := FALSE, Test := _Assertions);

	E_RunPhase.Teardown:
		_Slot.Teardown.Teardown(Enable := FALSE, Test := _Assertions);
END_CASE

_PhaseDeadline.Disarm();
// Errored, not Failed and not Skipped. The code under test was never shown to be

// wrong, and a Skipped verdict must not turn a build red - but an abandoned run

// must not read as a clean one either.
IF _Journal.Status = E_TestStatus.Running THEN
	_Journal.RecordFailure(Kind := E_FailureKind.Environment, Diagnostic := 'abandoned before completing', Message := '');
	_Journal.Finish(E_TestStatus.Errored);
END_IF

THIS^.Unload();
_Outcome := E_PhaseOutcome.Finished;
END_METHOD

// The label of the test most recently loaded. Survives Unload deliberately.

//

// The suite raises its framework error for a teardown overrun on the scan AFTER

// the runner unloaded, so a label cleared at Unload would leave that error naming

// nothing. Empty only before the first Load.
PROPERTY ActiveLabel : T_MaxString
GET
ActiveLabel := _LastLabel;
END_GET
END_PROPERTY

// One scan of the active test. Call every scan while the suite is enabled.

//

// Enable is held, not edged: it is passed straight through to whichever phase is

// running. Dropping it abandons the test - the phase in flight gets one final

// call with Enable FALSE so it can put its own state back, and its return value

// is ignored, because a test that failed by hanging will not answer that call

// either.
METHOD Advance : E_PhaseOutcome
VAR_INPUT
	Enable : BOOL;
END_VAR

VAR
	PhaseDone : BOOL;
END_VAR
Advance := _Outcome;
IF _Outcome <> E_PhaseOutcome.Running THEN
	// A TERMINAL OUTCOME IS REPORTED EXACTLY ONCE, on the scan it happens - the

	// CASE below returns it directly. Every call after that says Idle.

	//

	// Returning the stored value again republishes the last test of the PREVIOUS

	// run: a re-run's first Advance happens before anything is loaded, so the suite

	// sees Finished, publishes _LastJournal, and records a case that already

	// existed. It never shows in a single run, because the suite stops calling once

	// complete - only a re-run reaches it, which is why CHAR_ReRunTests is the only

	// thing that found it.

	//

	// The Outcome PROPERTY still reports the real terminal value for anyone
	// inspecting the runner; it is only the driving call that goes quiet.
	Advance := E_PhaseOutcome.Idle;
	RETURN;
END_IF

IF NOT Enable THEN
	THIS^.Abandon();
	Advance := _Outcome;
	RETURN;
END_IF

CASE _Phase OF
	E_RunPhase.Setup:
		PhaseDone := _Slot.Setup.Setup(Enable := TRUE, Test := _Assertions);
		IF PhaseDone THEN
			_PhaseDeadline.Disarm();
			// A failure or error recorded during setup ends the test WITHOUT running the

			// body. A test whose fixture never came up has not been exercised, and

			// reporting it as a failed check would be a lie.

			//

			// Kind is what answers this, not Status: RecordFailure does not move the

			// journal out of Running - only Complete does - so Status is still Running

			// here whatever setup found. Kind is None until a failure is recorded.
			IF _Journal.Kind <> E_FailureKind.None THEN
				_Journal.Finish(E_TestStatus.Failed);
				THIS^.BeginTeardown();
			ELSE
				_Phase := E_RunPhase.Body;
			END_IF
		ELSIF _PhaseDeadline.Tick() THEN
			_Journal.RecordFailure(Kind := E_FailureKind.Timeout, Diagnostic := _PhaseDeadline.Diagnostic, Message := '');
			_Journal.Finish(E_TestStatus.Failed);
			THIS^.BeginTeardown();
		END_IF

	E_RunPhase.Body:
		PhaseDone := _Slot.Test.Run(Enable := TRUE, Test := _Assertions);
		IF PhaseDone THEN
			_Journal.Finish(E_TestStatus.Passed);
			THIS^.BeginTeardown();
		ELSIF _Journal.Tick() THEN
			// Tick recorded the timeout and finished the journal itself.
			THIS^.BeginTeardown();
		END_IF

	E_RunPhase.Teardown:
		PhaseDone := _Slot.Teardown.Teardown(Enable := TRUE, Test := _Assertions);
		IF PhaseDone THEN
			_PhaseDeadline.Disarm();
			THIS^.Unload();
			_Outcome := E_PhaseOutcome.Finished;
		ELSIF _PhaseDeadline.Tick() THEN
			// Abandoned, not failed. The verdict stands: a passing test whose cleanup

			// hung still proved the code correct. The suite raises a framework error and
			// the run goes red.
			_TeardownDiagnostic := _PhaseDeadline.Diagnostic;
			THIS^.Unload();
			_Outcome := E_PhaseOutcome.TeardownOverran;
		END_IF
END_CASE

Advance := _Outcome;
END_METHOD

// Wire the runner up. Called once by the suite at composition.

//

// The verdict handle is one per suite and is retargeted here, per test, because

// only one test runs at a time. At capacity 50 that is one copy of the assertion

// machinery rather than fifty.
METHOD Attach
VAR_INPUT
	Roster : I_TestRoster;
END_VAR

VAR_IN_OUT
	Verdict : TestVerdict;
END_VAR
_Roster		:= Roster;
_Verdict	REF= Verdict;
_Assertions := Verdict;
END_METHOD

// Move to teardown, or finish if there is none.

//

// Teardown runs whatever the verdict - passed, failed, errored, timed out. This is

// a guarantee only reachable because the runner calls the tests rather than

// so could not call anything after them.

//

// Its deadline is its own and is usually shorter than the body's. A test that

// failed by hanging is now being asked to clean up and will most likely hang

// again, and on a rig that means an axis left powered.
METHOD BeginTeardown
VAR
	Budgets : ST_TestBudgets;
END_VAR
// The journal must be terminal before teardown reads Status to decide how to

// clean up. Setup failure and body completion both leave it so; this covers the
// path where neither did.
IF _Journal.Status = E_TestStatus.Running THEN
	_Journal.Finish(E_TestStatus.Passed);
END_IF

IF _Slot.Teardown = 0 THEN
	THIS^.Unload();
	_Outcome := E_PhaseOutcome.Finished;
	RETURN;
END_IF

Budgets := _Journal.Budgets;
_Phase	:= E_RunPhase.Teardown;
_PhaseDeadline.Arm('teardown', Budgets.Teardown);
END_METHOD

// Make this slot the active test and start it. One call, then Advance every scan

// until it stops returning Running.

//

// Begin is called BEFORE setup so the wall clock covers the whole test. The

// journal is ticked only while the BODY runs, so ElapsedCycles - and therefore

// AssertCompletedWithin - measure the body rather than the fixture, and

// IsFirstCycle is TRUE on the body's first scan as documented.

//

// Returns FALSE if the slot carries no test or the runner is not attached, in

// which case nothing is loaded and Outcome stays Idle.
METHOD Load : BOOL
VAR_INPUT
	Slot : ST_TestSlot;
END_VAR

VAR
	Location : T_MaxString;

	// A property returning a STRUCT cannot have a member read off the call result.

	// It is copied to a local first - a TwinCAT rule, not a style choice.
	Budgets : ST_TestBudgets;
END_VAR
Load := FALSE;
IF (Slot.Test = 0) OR (_Roster = 0) OR NOT __ISVALIDREF(_Verdict) THEN
	RETURN;
END_IF

_Slot	   := Slot;
_LastLabel := Slot.Label;
_Journal   REF= _Roster.Journal(Slot.Index);
IF NOT __ISVALIDREF(_Journal) THEN
	// The slot and the roster disagree. Running nothing is safer than writing
	// through an invalid reference.
	_Slot	 := _EmptySlot;
	_Outcome := E_PhaseOutcome.Idle;
	RETURN;
END_IF

IF _Slot.Location <> 0 THEN
	Location := _Slot.Location.Path;
END_IF

_Journal.Begin(Label := _Slot.Label, Location := Location);
_Verdict.Target(_Journal);

// Setup is skipped entirely by a test that does not implement it. There is no

// empty method body to call and no flag to keep in step.
Budgets := _Journal.Budgets;
IF _Slot.Setup <> 0 THEN
	_Phase := E_RunPhase.Setup;
	_PhaseDeadline.Arm('setup', Budgets.Setup);
ELSE
	_Phase := E_RunPhase.Body;
END_IF

_Outcome := E_PhaseOutcome.Running;
Load	 := TRUE;
END_METHOD

// What the last Advance did. Idle when nothing is loaded.
PROPERTY Outcome : E_PhaseOutcome
GET
Outcome := _Outcome;
END_GET
END_PROPERTY

// Why teardown was abandoned, for the framework error the suite raises. Empty

// unless the last Advance returned TeardownOverran.
PROPERTY TeardownDiagnostic : T_MaxString
GET
TeardownDiagnostic := _TeardownDiagnostic;
END_GET
END_PROPERTY

// Drop the active test. The verdict handle is untargeted so a stray call cannot

// write into a finished test's record.
METHOD Unload
_Verdict.Untarget();
_Journal REF= 0;
_Slot	 := _EmptySlot;
_Phase	 := E_RunPhase.Idle;
END_METHOD

END_FUNCTION_BLOCK

// ---- POUs/TestVerdict.TcPOU
// The handle a test body reports through - the object passed as the Test

// parameter of I_Test.Run.

//

// ONE instance per suite, not one per test. Only one test runs at a time, so the

// handle is retargeted to whichever journal is active rather than allocated per

// slot. At capacity 50 that is the difference between one copy of the assertion

// machinery and fifty. Allocating all of it per slot is most of

// why a referencing project paid for it whether it ran tests or not.

//

// Its single job is turning a check into a record: dispatch the comparison,

// compose the diagnostic, count it in the journal and stream it to the detail

// sink. The comparing itself belongs to TestValueCompare, which is pure and

// testable on its own.

//

// Being one per suite is what makes it the right place to hold the detail sink:

// every check in the suite already passes through here, so the sink is one

// reference rather than one per slot.
FUNCTION_BLOCK TestVerdict IMPLEMENTS I_TestAssertions
VAR
	_Journal	: REFERENCE TO TestJournal;
	_DetailSink : I_TestDetailSink;
END_VAR

(*
	No cyclic body. Every entry point is driven by a check in a test body.
*)

// Lengths first, so a size difference is reported as one rather than as a

// difference at whatever byte happens to differ.
METHOD AssertBufferEqual
VAR_INPUT
	pExpected	   : POINTER TO BYTE;
	ExpectedLength : UDINT;
	pActual		   : POINTER TO BYTE;
	ActualLength   : UDINT;
	Message		   : T_MaxString;
END_VAR

VAR
	ExpectedText : T_MaxString;
	ActualText	 : T_MaxString;
END_VAR
IF ExpectedLength <> ActualLength THEN
	// Lengths first, so a size difference is reported as one rather than as a
	// difference at whatever byte happens to differ.
	ExpectedText := CONCAT(LREAL_TO_FMTSTR(TO_LREAL(ExpectedLength), 0, FALSE), ' bytes');
	ActualText	 := CONCAT(LREAL_TO_FMTSTR(TO_LREAL(ActualLength), 0, FALSE), ' bytes');
	THIS^.Emit(Kind		  := E_FailureKind.SizeMismatch,
			   Expected	  := ExpectedText,
			   Actual	  := ActualText,
			   Diagnostic := CONCAT(CONCAT(CONCAT('expected ', ExpectedText), ', actual '), ActualText),
			   Message	  := Message);

	RETURN;
END_IF

THIS^.AssertMemEqual(pExpected,
					 pActual,
					 ExpectedLength,
					 Message);
END_METHOD

// Compares against COMPLETED scans: the one in progress is not counted, because

// the journal is ticked after the body runs. See I_TestTiming.ElapsedCycles.

//

// Opt-in, never a default. A scan budget is a real regression signal on a fixed

// target and noise across a matrix of them.
METHOD AssertCompletedWithin
VAR_INPUT
	Cycles	: UDINT;
	Message : T_MaxString;
END_VAR

VAR
	ExpectedText : T_MaxString;
	ActualText	 : T_MaxString;
END_VAR
IF NOT __ISVALIDREF(_Journal) THEN
	RETURN;
END_IF

IF _Journal.ElapsedCycles <= Cycles THEN
	THIS^.RecordPass(Message);
	RETURN;
END_IF

ExpectedText := CONCAT(CONCAT('within ', LREAL_TO_FMTSTR(TO_LREAL(Cycles), 0, FALSE)), ' cycles');
ActualText	 := CONCAT(LREAL_TO_FMTSTR(TO_LREAL(_Journal.ElapsedCycles), 0, FALSE), ' cycles');
THIS^.Emit(Kind		  := E_FailureKind.Timeout,
		   Expected	  := ExpectedText,
		   Actual	  := ActualText,
		   Diagnostic := CONCAT(CONCAT(CONCAT('expected ', ExpectedText), ', actual '), ActualText),
		   Message	  := Message);
END_METHOD

// See TestValueCompare for what equality means here - notably that REAL and

// LREAL compare exactly, and that a size difference is its own failure kind.
METHOD AssertEqual
VAR_INPUT
	Expected : ANY;
	Actual	 : ANY;
	Message	 : T_MaxString;
END_VAR

VAR
	Comparison : ST_CompareResult;
END_VAR
Comparison := TestValueCompare(Expected, Actual);
IF Comparison.IsEqual THEN
	THIS^.RecordPass(Message);
ELSE
	THIS^.Emit(Kind		  := Comparison.Kind,
			   Expected	  := Comparison.Expected,
			   Actual	  := Comparison.Actual,
			   Diagnostic := Comparison.Diagnostic,
			   Message	  := Message);
END_IF
END_METHOD

METHOD AssertFalse
VAR_INPUT
	Condition : BOOL;
	Message	  : T_MaxString;
END_VAR
IF NOT Condition THEN
	THIS^.RecordPass(Message);
ELSE
	THIS^.Emit(Kind		  := E_FailureKind.ValueMismatch,
			   Expected	  := 'FALSE',
			   Actual	  := 'TRUE',
			   Diagnostic := 'expected FALSE, actual TRUE',
			   Message	  := Message);
END_IF
END_METHOD

METHOD AssertGreater
VAR_INPUT
	Actual	: ANY;
	Bound	: ANY;
	Message : T_MaxString;
END_VAR

VAR
	ActualNumber : ST_NumericValue;
	BoundNumber	 : ST_NumericValue;
	ExpectedText : T_MaxString;
	ActualText	 : T_MaxString;
END_VAR
ActualNumber := TestValueAsLReal(Actual);
BoundNumber	 := TestValueAsLReal(Bound);
IF NOT (ActualNumber.IsNumeric AND BoundNumber.IsNumeric) THEN
	THIS^.RecordFailure(E_FailureKind.TypeMismatch, 'not an ordered type', Message);
ELSIF ActualNumber.Value > BoundNumber.Value THEN
	THIS^.RecordPass(Message);
ELSE
	ExpectedText := CONCAT('greater than ', TestValueString(Bound));
	ActualText	 := TestValueString(Actual);
	THIS^.Emit(Kind		  := E_FailureKind.ValueMismatch,
			   Expected	  := ExpectedText,
			   Actual	  := ActualText,
			   Diagnostic := CONCAT(CONCAT(CONCAT('expected ', TestValueBrief(ExpectedText)), ', actual '), TestValueBrief(ActualText)),
			   Message	  := Message);
END_IF
END_METHOD

METHOD AssertInRange
VAR_INPUT
	Actual	: LREAL;
	Minimum : LREAL;
	Maximum : LREAL;
	Message : T_MaxString;
END_VAR

VAR
	ExpectedText : T_MaxString;
	ActualText	 : T_MaxString;
END_VAR
IF (Actual >= Minimum) AND (Actual <= Maximum) THEN
	THIS^.RecordPass(Message);
	RETURN;
END_IF

ExpectedText := CONCAT(CONCAT(LREAL_TO_FMTSTR(Minimum, 6, TRUE), ' to '), LREAL_TO_FMTSTR(Maximum, 6, TRUE));
ActualText	 := LREAL_TO_FMTSTR(Actual, 6, TRUE);
THIS^.Emit(Kind		  := E_FailureKind.ValueMismatch,
		   Expected	  := ExpectedText,
		   Actual	  := ActualText,
		   Diagnostic := CONCAT(CONCAT(CONCAT('expected ', ExpectedText), ', actual '), ActualText),
		   Message	  := Message);
END_METHOD

PROPERTY AssertionCount : UDINT
GET
IF __ISVALIDREF(_Journal) THEN
	AssertionCount := _Journal.AssertionCount;
END_IF
END_GET
END_PROPERTY

METHOD AssertLess
VAR_INPUT
	Actual	: ANY;
	Bound	: ANY;
	Message : T_MaxString;
END_VAR

VAR
	ActualNumber : ST_NumericValue;
	BoundNumber	 : ST_NumericValue;
	ExpectedText : T_MaxString;
	ActualText	 : T_MaxString;
END_VAR
ActualNumber := TestValueAsLReal(Value := Actual);
BoundNumber	 := TestValueAsLReal(Value := Bound);
IF NOT (ActualNumber.IsNumeric AND BoundNumber.IsNumeric) THEN
	THIS^.RecordFailure(E_FailureKind.TypeMismatch, 'not an ordered type', Message);
ELSIF ActualNumber.Value < BoundNumber.Value THEN
	THIS^.RecordPass(Message);
ELSE
	ExpectedText := CONCAT('less than ', TestValueString(Bound));
	ActualText	 := TestValueString(Actual);
	THIS^.Emit(Kind		  := E_FailureKind.ValueMismatch,
			   Expected	  := ExpectedText,
			   Actual	  := ActualText,
			   Diagnostic := CONCAT(CONCAT(CONCAT('expected ', TestValueBrief(ExpectedText)), ', actual '), TestValueBrief(ActualText)),
			   Message	  := Message);
END_IF
END_METHOD

METHOD AssertMemEqual
VAR_INPUT
	pExpected : POINTER TO BYTE;
	pActual	  : POINTER TO BYTE;
	Length	  : UDINT;
	Message	  : T_MaxString;
END_VAR

VAR
	pLeft		 : POINTER TO BYTE;
	pRight		 : POINTER TO BYTE;
	i			 : DINT;
	ExpectedText : T_MaxString;
	ActualText	 : T_MaxString;
END_VAR
IF (pExpected = 0) OR (pActual = 0) THEN
	// Environment, not ValueMismatch: nothing was compared, so nothing about the
	// code under test was shown to be wrong. No values to report either.
	THIS^.RecordFailure(E_FailureKind.Environment, 'null buffer', Message);
	RETURN;
END_IF

pLeft  := pExpected;
pRight := pActual;
FOR i := 0 TO TO_DINT(Length) - 1 DO
	IF pLeft[i] <> pRight[i] THEN
		ExpectedText := CONCAT('16#', BYTE_TO_HEXSTR(pLeft[i], 2, TRUE));
		ActualText	 := CONCAT('16#', BYTE_TO_HEXSTR(pRight[i], 2, TRUE));
		THIS^.Emit(Kind		  := E_FailureKind.ValueMismatch,
				   Expected	  := ExpectedText,
				   Actual	  := ActualText,
				   Diagnostic := CONCAT(CONCAT(CONCAT(CONCAT(CONCAT('differs at byte ', LREAL_TO_FMTSTR(TO_LREAL(i), 0, FALSE)), ': expected '), ExpectedText), ', actual '), ActualText),
				   Message	  := Message);

		RETURN;
	END_IF
END_FOR

THIS^.RecordPass(Message);
END_METHOD

// ABSOLUTE tolerance: passes when |Expected - Actual| <= Tolerance.

//

// Tolerance carries the units of the value being compared - millimetres, volts,

// encoder counts. Use it when you know how much error is acceptable in those

// units, which is usually true of a physical measurement.

//

// At large magnitudes an absolute tolerance can fall below what an LREAL can

// represent, at which point it degenerates into exact equality. AssertWithin does

// not have that problem.
METHOD AssertNear
VAR_INPUT
	Expected  : LREAL;
	Actual	  : LREAL;
	Tolerance : LREAL;
	Message	  : T_MaxString;
END_VAR

VAR
	ExpectedText : T_MaxString;
	ActualText	 : T_MaxString;
END_VAR
IF ABS(Expected - Actual) <= ABS(Tolerance) THEN
	THIS^.RecordPass(Message);
	RETURN;
END_IF

// The tolerance belongs with the expectation, not beside it: what the test

// demanded is a band, and a reader comparing 5.000000 with 5.002000 cannot see

// whether that was meant to pass without it.
ExpectedText := CONCAT(CONCAT(CONCAT(LREAL_TO_FMTSTR(Expected, 6, TRUE), ' +/- '), LREAL_TO_FMTSTR(ABS(Tolerance), 6, TRUE)), '');
ActualText	 := LREAL_TO_FMTSTR(Actual, 6, TRUE);
THIS^.Emit(Kind		  := E_FailureKind.ValueMismatch,
		   Expected	  := ExpectedText,
		   Actual	  := ActualText,
		   Diagnostic := CONCAT(CONCAT(CONCAT('expected ', ExpectedText), ', actual '), ActualText),
		   Message	  := Message);
END_METHOD

METHOD AssertNotEqual
VAR_INPUT
	Expected : ANY;
	Actual	 : ANY;
	Message	 : T_MaxString;
END_VAR

VAR
	Comparison : ST_CompareResult;
	Rendered   : T_MaxString;
END_VAR
Comparison := TestValueCompare(Expected, Actual);
IF NOT Comparison.IsEqual THEN
	THIS^.RecordPass(Message);
ELSE
	Rendered := TestValueString(Expected);
	THIS^.Emit(Kind		  := E_FailureKind.ValueMismatch,
			   Expected	  := CONCAT('any value other than ', Rendered),
			   Actual	  := Rendered,
			   Diagnostic := CONCAT('expected any value other than ', TestValueBrief(Rendered)),
			   Message	  := Message);
END_IF
END_METHOD

METHOD AssertTrue
VAR_INPUT
	Condition : BOOL;
	Message	  : T_MaxString;
END_VAR
IF Condition THEN
	THIS^.RecordPass(Message);
ELSE
	THIS^.Emit(Kind		  := E_FailureKind.ValueMismatch,
			   Expected	  := 'TRUE',
			   Actual	  := 'FALSE',
			   Diagnostic := 'expected TRUE, actual FALSE',
			   Message	  := Message);
END_IF
END_METHOD

// RELATIVE tolerance: passes when |Expected - Actual| <= |Expected| * Fraction.

//

// Holds its meaning across magnitudes, which absolute tolerance does not - 0.1 per

// cent means the same thing at 1.0 and at 1E9. Use it for ratios, gains, scaled

// values, and anywhere the acceptable error scales with the value itself.

//

// Near zero it collapses: |Expected| * Fraction approaches nothing, so an expected

// value of zero admits only an exact match. That is not a defect to paper over

// with a hidden floor - if zero is the expected value, an absolute tolerance is

// what the situation calls for, and AssertNear is the method that expresses it.
METHOD AssertWithin
VAR_INPUT
	Expected : LREAL;
	Actual	 : LREAL;

	// Dimensionless. 0.001 is 0.1 per cent of Expected.
	Fraction : LREAL;
	Message	 : T_MaxString;
END_VAR

VAR
	Tolerance	 : LREAL;
	ExpectedText : T_MaxString;
	ActualText	 : T_MaxString;
END_VAR
Tolerance := ABS(Expected) * ABS(Fraction);
IF ABS(Expected - Actual) <= Tolerance THEN
	THIS^.RecordPass(Message);
	RETURN;
END_IF

ActualText := LREAL_TO_FMTSTR(Actual, 6, TRUE);
IF Expected = 0.0 THEN
	// A relative tolerance around zero admits only zero. Say which method the
	// situation actually calls for rather than reporting a mysterious near miss.
	ExpectedText := 'exactly 0 (relative tolerance admits nothing else - use AssertNear)';
	THIS^.Emit(Kind		  := E_FailureKind.ValueMismatch,
			   Expected	  := ExpectedText,
			   Actual	  := ActualText,
			   Diagnostic := CONCAT(CONCAT('expected ', ExpectedText), CONCAT(', actual ', ActualText)),
			   Message	  := Message);

	RETURN;
END_IF

// Both forms of the band: the fraction the author wrote, and what it works out to

// at this magnitude. Either one alone leaves the reader doing arithmetic.
ExpectedText := LREAL_TO_FMTSTR(Expected, 6, TRUE);
ExpectedText := CONCAT(ExpectedText, ' +/- ');
ExpectedText := CONCAT(ExpectedText, LREAL_TO_FMTSTR(ABS(Fraction) * 100.0, 4, TRUE));
ExpectedText := CONCAT(ExpectedText, '% (');
ExpectedText := CONCAT(ExpectedText, LREAL_TO_FMTSTR(Tolerance, 6, TRUE));
ExpectedText := CONCAT(ExpectedText, ')');
THIS^.Emit(Kind		  := E_FailureKind.ValueMismatch,
		   Expected	  := ExpectedText,
		   Actual	  := ActualText,
		   Diagnostic := CONCAT(CONCAT('expected ', ExpectedText), CONCAT(', actual ', ActualText)),
		   Message	  := Message);
END_METHOD

// Where individual checks go. Called once by the suite at composition; a null sink

// is the normal case and costs one comparison per check.

//

// Not on I_TestAssertions. A test body holds this object and must not be able to

// redirect the record of its own run.
METHOD AttachDetailSink
VAR_INPUT
	Sink : I_TestDetailSink;
END_VAR
_DetailSink := Sink;
END_METHOD

PROPERTY ElapsedCycles : UDINT
GET
IF __ISVALIDREF(_Journal) THEN
	ElapsedCycles := _Journal.ElapsedCycles;
END_IF
END_GET
END_PROPERTY

PROPERTY ElapsedTime : LREAL
GET
IF __ISVALIDREF(_Journal) THEN
	ElapsedTime := _Journal.ElapsedTime;
END_IF
END_GET
END_PROPERTY

// The one place a failure becomes a record. Private: I_TestOutcome.RecordFailure

// is the public door and delegates here with no values.

//

// Kept private rather than widening RecordFailure because that method is the

// narrow type domain helpers take. An NC helper reporting that an axis never

// homed has no expected-and-actual pair, and should not be made to pass two empty

// strings to say so.
METHOD Emit
VAR_INPUT
	Kind : E_FailureKind;

	// Full rendered values, or empty when the failure has no two values.
	Expected   : T_MaxString;
	Actual	   : T_MaxString;
	Diagnostic : T_MaxString;
	Message	   : T_MaxString;
END_VAR

VAR
	StepLabel : T_MaxString;
END_VAR
IF NOT __ISVALIDREF(_Journal) THEN
	RETURN;
END_IF

// The step is read before the journal records anything, so a streamed check

// carries the step it actually ran under.
StepLabel := _Journal.StepLabel;
_Journal.RecordFailure(Kind, Diagnostic, Message);
IF _DetailSink <> 0 THEN
	_DetailSink.CheckFailed(StepLabel  := StepLabel,
							Kind	   := Kind,
							Expected   := Expected,
							Actual	   := Actual,
							Diagnostic := Diagnostic,
							Message	   := Message);
END_IF
END_METHOD

METHOD Fail
VAR_INPUT
	Reason : T_MaxString;
END_VAR
THIS^.RecordFailure(E_FailureKind.ValueMismatch, 'explicit failure', Reason);
END_METHOD

PROPERTY IsFirstCycle : BOOL
GET
IF __ISVALIDREF(_Journal) THEN
	IsFirstCycle := _Journal.IsFirstCycle;
END_IF
END_GET
END_PROPERTY

METHOD RecordFailure
VAR_INPUT
	Kind	   : E_FailureKind;
	Diagnostic : T_MaxString;
	Message	   : T_MaxString;
END_VAR
THIS^.Emit(Kind		  := Kind,
		   Expected	  := '',
		   Actual	  := '',
		   Diagnostic := Diagnostic,
		   Message	  := Message);
END_METHOD

METHOD RecordPass
VAR_INPUT
	Detail : T_MaxString;
END_VAR
IF NOT __ISVALIDREF(_Journal) THEN
	RETURN;
END_IF

_Journal.RecordPass();
IF _DetailSink <> 0 THEN
	_DetailSink.CheckPassed(StepLabel := _Journal.StepLabel, Detail := Detail);
END_IF
END_METHOD

METHOD ReportError
VAR_INPUT
	Reason : T_MaxString;
END_VAR
THIS^.RecordFailure(E_FailureKind.Environment, 'could not run', Reason);
END_METHOD

METHOD SetStep
VAR_INPUT
	Label : T_MaxString;
END_VAR
IF __ISVALIDREF(_Journal) THEN
	_Journal.SetStep(Label);
END_IF
END_METHOD

PROPERTY Status : E_TestStatus
GET
IF __ISVALIDREF(_Journal) THEN
	Status := _Journal.Status;
ELSE
	Status := E_TestStatus.NotStarted;
END_IF
END_GET
END_PROPERTY

// Point the handle at the active test's journal. Called by the suite, never by a

// test.
METHOD Target
VAR_INPUT
	Journal : REFERENCE TO TestJournal;
END_VAR
_Journal REF= Journal;
END_METHOD

// Point the handle at nothing. Called by the runner when a test finishes, so a

// stray call cannot write into a completed test's record - or worse, into the

// next test's.

//

// Every method here already guards on __ISVALIDREF, so an untargeted handle is

// inert rather than dangerous. This is what makes that guard mean something.
METHOD Untarget
_Journal REF= 0;
END_METHOD

END_FUNCTION_BLOCK

// ---- POUs/TestValueCompare.TcPOU
// Compares any two values and says whether they match, and if not, why.

//

// Pure: no state, no reporting, no verdict. That makes it the one part of the

// framework testable in isolation - including against the OLD library, before the

// new runner exists.

//

// WHAT IS BEING TESTED decides the rule. A test author writing AssertEqual is

// testing a value, so the storage that value happens to sit in is not the subject:

//

//   strings   compared by CONTENT. Declared capacity is ignored - STRING(20) and

//             STRING(80) holding 'homed' are equal. diSize for a string is the

//             capacity of the variable, not the length of the value, so comparing

//             it would be testing the declaration. If capacity or length is the

//             subject, say so: AssertEqual(ExpectedLength, LEN(Actual)).

//

//   numerics  compared by VALUE across widths. INT#5 equals DINT#5. The width is

//             incidental to what the author is checking.

//

//   the rest  structs, arrays, times, enums: compared by size, then by bytes. A

//             size difference here is a genuine TypeMismatch - different types

//             rather than different values.

//

// Two rules worth stating outright:

//

//  1. WSTRING is compared AS WSTRING, not by copying its bytes into a

//     STRING buffer and compared with '<>', which terminates at the first NUL -

//     and every second byte of ASCII WSTRING content is NUL. Two different

//     WSTRINGs of equal declared size compared equal and the test went green.

//

//  2. REAL and LREAL compare EXACTLY, with no hidden epsilon of

//     0.000001, so a test passing at 1E-7 looked identical to one passing exactly.

//     Tolerance now has its own methods - AssertNear for absolute, AssertWithin

//     for relative - and choosing one is visible at the call site.

//

//     Because exact float equality is a classic trap, a near-miss on a float

//     appends a hint naming the two methods.
FUNCTION TestValueCompare : ST_CompareResult
VAR_INPUT
	Expected : ANY;
	Actual	 : ANY;
END_VAR

VAR
	ExpectedText   : T_MaxString;
	ActualText	   : T_MaxString;
	ExpectedWide   : WSTRING(255);
	ActualWide	   : WSTRING(255);
	ExpectedNumber : ST_NumericValue;
	ActualNumber   : ST_NumericValue;
	pExpected	   : POINTER TO BYTE;
	pActual		   : POINTER TO BYTE;
	i			   : DINT;
	Spread		   : LREAL;
END_VAR

VAR CONSTANT
	// Only ever used to decide whether to SUGGEST a tolerance method. Never

	// applied as one.
	HintThreshold : LREAL := 1E-6;
END_VAR

TestValueCompare.IsEqual	:= FALSE;
TestValueCompare.Kind		:= E_FailureKind.ValueMismatch;
TestValueCompare.Diagnostic := '';
TestValueCompare.Expected	:= '';
TestValueCompare.Actual		:= '';
// ---- strings: content only ------------------------------------------------
IF TestValueIsText(Expected) AND TestValueIsText(Actual) THEN
	// WSTRING is converted, never reinterpreted. Comparing its bytes as a STRING
	// stops at the first character.
	IF Expected.TypeClass = __SYSTEM.TYPE_CLASS.TYPE_WSTRING THEN
		MEMCPY(ADR(ExpectedWide), Expected.pValue, MIN(SIZEOF(ExpectedWide), TO_UDINT(Expected.diSize)));
		WSTRING_TO_STRING2(ADR(ExpectedText), ADR(ExpectedWide), SIZEOF(ExpectedText));
	ELSE
		MEMCPY(ADR(ExpectedText), Expected.pValue, MIN(SIZEOF(ExpectedText), TO_UDINT(Expected.diSize)));
	END_IF

	IF Actual.TypeClass = __SYSTEM.TYPE_CLASS.TYPE_WSTRING THEN
		MEMCPY(ADR(ActualWide), Actual.pValue, MIN(SIZEOF(ActualWide), TO_UDINT(Actual.diSize)));
		WSTRING_TO_STRING2(ADR(ActualText), ADR(ActualWide), SIZEOF(ActualText));
	ELSE
		MEMCPY(ADR(ActualText), Actual.pValue, MIN(SIZEOF(ActualText), TO_UDINT(Actual.diSize)));
	END_IF

	IF ExpectedText = ActualText THEN
		TestValueCompare.IsEqual := TRUE;
		TestValueCompare.Kind	 := E_FailureKind.None;
	ELSE
		TestValueCompare.Expected	:= TestValueString(Expected);
		TestValueCompare.Actual		:= TestValueString(Actual);
		TestValueCompare.Diagnostic := CONCAT(CONCAT(CONCAT('expected ', TestValueBrief(TestValueCompare.Expected)), ', actual '), TestValueBrief(TestValueCompare.Actual));
	END_IF

	RETURN;
END_IF

// ---- numerics: value across widths ----------------------------------------
ExpectedNumber := TestValueAsLReal(Expected);
ActualNumber   := TestValueAsLReal(Actual);
IF ExpectedNumber.IsNumeric AND ActualNumber.IsNumeric THEN
	IF ExpectedNumber.Value = ActualNumber.Value THEN
		TestValueCompare.IsEqual := TRUE;
		TestValueCompare.Kind	 := E_FailureKind.None;
		RETURN;
	END_IF

	TestValueCompare.Expected	:= TestValueString(Expected);
	TestValueCompare.Actual		:= TestValueString(Actual);
	TestValueCompare.Diagnostic := CONCAT(CONCAT(CONCAT('expected ', TestValueBrief(TestValueCompare.Expected)), ', actual '), TestValueBrief(TestValueCompare.Actual));
	// A near miss on a float is almost always someone expecting tolerance from

	// exact equality. Say so where they are already looking.
	IF TestValueIsFloat(Expected) OR TestValueIsFloat(Actual) THEN
		Spread := ABS(ExpectedNumber.Value - ActualNumber.Value);
		IF Spread <= (HintThreshold * MAX(1.0, ABS(ExpectedNumber.Value))) THEN
			TestValueCompare.Diagnostic := CONCAT(TestValueCompare.Diagnostic, ' (use AssertNear or AssertWithin for floats)');
		END_IF
	END_IF

	RETURN;
END_IF

// ---- one numeric, one not -------------------------------------------------
IF ExpectedNumber.IsNumeric <> ActualNumber.IsNumeric THEN
	TestValueCompare.Kind		:= E_FailureKind.TypeMismatch;
	TestValueCompare.Diagnostic := 'compared a numeric value with a non-numeric one';
	RETURN;
END_IF

// ---- everything else: size, then bytes ------------------------------------

// Structs, arrays, times, enums. Here a size difference IS a type difference,

// not two spellings of the same value.
IF Expected.diSize <> Actual.diSize THEN
	TestValueCompare.Kind		:= E_FailureKind.TypeMismatch;
	TestValueCompare.Expected	:= CONCAT(LREAL_TO_FMTSTR(TO_LREAL(Expected.diSize), 0, FALSE), ' bytes');
	TestValueCompare.Actual		:= CONCAT(LREAL_TO_FMTSTR(TO_LREAL(Actual.diSize), 0, FALSE), ' bytes');
	TestValueCompare.Diagnostic := CONCAT(CONCAT(CONCAT('expected ', TestValueCompare.Expected), ', actual '), TestValueCompare.Actual);
	RETURN;
END_IF

pExpected := Expected.pValue;
pActual	  := Actual.pValue;
FOR i := 0 TO TO_DINT(Expected.diSize) - 1 DO
	IF pExpected[i] <> pActual[i] THEN
		TestValueCompare.Expected	:= TestValueString(Expected);
		TestValueCompare.Actual		:= TestValueString(Actual);
		TestValueCompare.Diagnostic := CONCAT(CONCAT(CONCAT(CONCAT(CONCAT('differs at byte ', LREAL_TO_FMTSTR(TO_LREAL(i), 0, FALSE)), ': expected '), TestValueBrief(TestValueCompare.Expected)), ', actual '), TestValueBrief(TestValueCompare.Actual));
		RETURN;
	END_IF
END_FOR

TestValueCompare.IsEqual := TRUE;
TestValueCompare.Kind	 := E_FailureKind.None;

END_FUNCTION

// ---- POUs/TestValueIsText.TcPOU
// TRUE for STRING and WSTRING.

//

// Split out so the rule lives in one place: 'is this a string' is asked by the

// comparison, by the formatter, and eventually by the reporters when they decide

// whether a value needs quoting.
FUNCTION TestValueIsText : BOOL
VAR_INPUT
	Value : ANY;
END_VAR

TestValueIsText := (Value.TypeClass = __SYSTEM.TYPE_CLASS.TYPE_STRING) OR (Value.TypeClass = __SYSTEM.TYPE_CLASS.TYPE_WSTRING);

END_FUNCTION

// ---- POUs/TestValueString.TcPOU
// Renders any value as text for a diagnostic.

//

// Returns T_MaxString, so a long value reaches the reporter intact and is

// shortened once, where the width is actually known.

//

// Unhandled type classes - enums, structs, arrays, pointers - render as hex bytes.

// Not friendly, but true: a diagnostic reading 'expected , actual ' tells the

// reader nothing at the moment they most need something.
FUNCTION TestValueString : T_MaxString
VAR_INPUT
	Value : ANY;
END_VAR

VAR
	Unsigned : ULINT;
	Signed8	 : SINT;
	Signed16 : INT;
	Signed32 : DINT;
	Signed64 : LINT;
	Real32	 : REAL;
	Real64	 : LREAL;
	Narrow	 : T_MaxString;
	Wide	 : WSTRING(255);
	ByteAt	 : POINTER TO BYTE;
	i		 : DINT;
	Shown	 : DINT;
END_VAR

TestValueString := '';
CASE Value.TypeClass OF
	__SYSTEM.TYPE_CLASS.TYPE_BOOL:
		MEMCPY(ADR(Unsigned), Value.pValue, TO_UDINT(Value.diSize));
		TestValueString := SEL(Unsigned <> 0, 'FALSE', 'TRUE');

	__SYSTEM.TYPE_CLASS.TYPE_BYTE, __SYSTEM.TYPE_CLASS.TYPE_USINT, __SYSTEM.TYPE_CLASS.TYPE_WORD, __SYSTEM.TYPE_CLASS.TYPE_UINT, __SYSTEM.TYPE_CLASS.TYPE_DWORD, __SYSTEM.TYPE_CLASS.TYPE_UDINT, __SYSTEM.TYPE_CLASS.TYPE_LWORD, __SYSTEM.TYPE_CLASS.TYPE_ULINT:
		MEMCPY(ADR(Unsigned), Value.pValue, TO_UDINT(Value.diSize));
		TestValueString := LREAL_TO_FMTSTR(TO_LREAL(Unsigned), 0, FALSE);

	__SYSTEM.TYPE_CLASS.TYPE_SINT:
		MEMCPY(ADR(Signed8), Value.pValue, TO_UDINT(Value.diSize));
		TestValueString := LREAL_TO_FMTSTR(TO_LREAL(Signed8), 0, FALSE);

	__SYSTEM.TYPE_CLASS.TYPE_INT:
		MEMCPY(ADR(Signed16), Value.pValue, TO_UDINT(Value.diSize));
		TestValueString := LREAL_TO_FMTSTR(TO_LREAL(Signed16), 0, FALSE);

	__SYSTEM.TYPE_CLASS.TYPE_DINT:
		MEMCPY(ADR(Signed32), Value.pValue, TO_UDINT(Value.diSize));
		TestValueString := LREAL_TO_FMTSTR(TO_LREAL(Signed32), 0, FALSE);

	__SYSTEM.TYPE_CLASS.TYPE_LINT:
		MEMCPY(ADR(Signed64), Value.pValue, TO_UDINT(Value.diSize));
		TestValueString := LREAL_TO_FMTSTR(TO_LREAL(Signed64), 0, FALSE);

	__SYSTEM.TYPE_CLASS.TYPE_REAL:
		MEMCPY(ADR(Real32), Value.pValue, TO_UDINT(Value.diSize));
		TestValueString := LREAL_TO_FMTSTR(TO_LREAL(Real32), 6, TRUE);

	__SYSTEM.TYPE_CLASS.TYPE_LREAL:
		MEMCPY(ADR(Real64), Value.pValue, TO_UDINT(Value.diSize));
		TestValueString := LREAL_TO_FMTSTR(Real64, 6, TRUE);

	__SYSTEM.TYPE_CLASS.TYPE_STRING:
		MEMCPY(ADR(Narrow), Value.pValue, MIN(SIZEOF(Narrow), TO_UDINT(Value.diSize)));
		TestValueString := CONCAT(CONCAT('$'', Narrow), '$'');

	__SYSTEM.TYPE_CLASS.TYPE_WSTRING:
		// Converted, never reinterpreted. Copying WSTRING bytes into a STRING

		// buffer terminates the text at the first character, because every second
		// byte of ASCII content is zero.
		MEMCPY(ADR(Wide), Value.pValue, MIN(SIZEOF(Wide), TO_UDINT(Value.diSize)));
		WSTRING_TO_STRING2(ADR(Narrow), ADR(Wide), SIZEOF(Narrow));
		TestValueString := CONCAT(CONCAT('$'', Narrow), '$'');

ELSE
	// Enums, structs, arrays, pointers, anything unrecognised. Hex is not
	// friendly, but it is true - and it beats an empty diagnostic.
	ByteAt			:= Value.pValue;
	Shown			:= MIN(TO_DINT(Value.diSize), 16);
	TestValueString := '16#';
	FOR i := 0 TO Shown - 1 DO
		TestValueString := CONCAT(TestValueString, BYTE_TO_HEXSTR(ByteAt[i], 2, TRUE));
	END_FOR

	IF TO_DINT(Value.diSize) > Shown THEN
		TestValueString := CONCAT(TestValueString, '...');
	END_IF
END_CASE

END_FUNCTION

// ---- POUs/TestValueBrief.TcPOU
// Shortens one rendered value to fit a composed line, with an ellipsis so the

// reader knows to look at the full value rather than believing this one.

//

// Exists because CONCAT cannot build a string longer than 255 characters at all -

// not merely because the destination is that wide. Two full values plus the words

// between them do not fit, so the composed diagnostic gets shortened copies and

// the full values travel separately in ST_CompareResult.

//

// Pure, and separate, because the budget arithmetic is the kind of thing that is

// wrong by one and never noticed.
FUNCTION TestValueBrief : T_MaxString
VAR_INPUT
	Value : T_MaxString;
END_VAR

VAR CONSTANT
	// The one place the budget exists. Two of these plus the longest surrounding

	// text - the byte-offset form, plus the float hint - stays inside 255, which is

	// the hard ceiling CONCAT itself imposes.

	//

	// Deliberately not a parameter. Every call site would then carry its own copy

	// of the number, which is the bug class Plan.md 2.1 names.
	Budget : INT := 80;
END_VAR

IF LEN(Value) <= TO_INT(Budget) THEN
	TestValueBrief := Value;
ELSE
	TestValueBrief := CONCAT(LEFT(Value, TO_INT(Budget - 3)), '...');
END_IF

END_FUNCTION

// ---- POUs/TestValueAsLReal.TcPOU
// Widens any numeric value to LREAL so ordering comparisons can be written once

// instead of per type.

//

// Returns ST_NumericValue rather than a value plus an output parameter.

// IsNumeric is FALSE for strings, structs, arrays and anything else with no

// ordering - the caller reports a TypeMismatch rather than comparing rubbish.

//

// LREAL carries 53 bits of mantissa, so LINT and ULINT values beyond 2^53 lose

// precision here. That matters for AssertGreater and AssertLess at extreme

// magnitudes and nowhere else; equality never goes through this path.
FUNCTION TestValueAsLReal : ST_NumericValue
VAR_INPUT
	Value : ANY;
END_VAR

VAR
	Unsigned : ULINT;
	Signed8	 : SINT;
	Signed16 : INT;
	Signed32 : DINT;
	Signed64 : LINT;
	Real32	 : REAL;
	Real64	 : LREAL;
END_VAR

TestValueAsLReal.Value	   := 0.0;
TestValueAsLReal.IsNumeric := TRUE;
CASE Value.TypeClass OF
	__SYSTEM.TYPE_CLASS.TYPE_BYTE, __SYSTEM.TYPE_CLASS.TYPE_USINT, __SYSTEM.TYPE_CLASS.TYPE_WORD, __SYSTEM.TYPE_CLASS.TYPE_UINT, __SYSTEM.TYPE_CLASS.TYPE_DWORD, __SYSTEM.TYPE_CLASS.TYPE_UDINT, __SYSTEM.TYPE_CLASS.TYPE_LWORD, __SYSTEM.TYPE_CLASS.TYPE_ULINT:
		MEMCPY(ADR(Unsigned), Value.pValue, TO_UDINT(Value.diSize));
		TestValueAsLReal.Value := TO_LREAL(Unsigned);

	__SYSTEM.TYPE_CLASS.TYPE_SINT:
		MEMCPY(ADR(Signed8), Value.pValue, TO_UDINT(Value.diSize));
		TestValueAsLReal.Value := TO_LREAL(Signed8);

	__SYSTEM.TYPE_CLASS.TYPE_INT:
		MEMCPY(ADR(Signed16), Value.pValue, TO_UDINT(Value.diSize));
		TestValueAsLReal.Value := TO_LREAL(Signed16);

	__SYSTEM.TYPE_CLASS.TYPE_DINT:
		MEMCPY(ADR(Signed32), Value.pValue, TO_UDINT(Value.diSize));
		TestValueAsLReal.Value := TO_LREAL(Signed32);

	__SYSTEM.TYPE_CLASS.TYPE_LINT:
		MEMCPY(ADR(Signed64), Value.pValue, TO_UDINT(Value.diSize));
		TestValueAsLReal.Value := TO_LREAL(Signed64);

	__SYSTEM.TYPE_CLASS.TYPE_REAL:
		MEMCPY(ADR(Real32), Value.pValue, TO_UDINT(Value.diSize));
		TestValueAsLReal.Value := TO_LREAL(Real32);

	__SYSTEM.TYPE_CLASS.TYPE_LREAL:
		MEMCPY(ADR(Real64), Value.pValue, TO_UDINT(Value.diSize));
		TestValueAsLReal.Value := Real64;

ELSE
	TestValueAsLReal.IsNumeric := FALSE;
END_CASE

END_FUNCTION

// ---- POUs/TestValueIsFloat.TcPOU
// TRUE for REAL and LREAL.

//

// Used only to decide whether a failed exact comparison deserves the hint about

// AssertNear and AssertWithin. Never used to apply a tolerance.
FUNCTION TestValueIsFloat : BOOL
VAR_INPUT
	Value : ANY;
END_VAR

TestValueIsFloat := (Value.TypeClass = __SYSTEM.TYPE_CLASS.TYPE_REAL) OR (Value.TypeClass = __SYSTEM.TYPE_CLASS.TYPE_LREAL);

END_FUNCTION

// ---- POUs/TestLogReporter.TcPOU
// Writes results to the TwinCAT system log through ADSLOGSTR.

//

// The simplest sink that is genuinely useful, and deliberately the first one

// built: it needs no project setup, no event class, and no asynchronous work, so

// attaching it cannot change whether a run completes. Anything that goes wrong

// here is visibly this object's fault and not the harness's.

//

// It implements I_TestReporter and NOT I_TestDetailSink. A log wants verdicts; a

// line per individual check would bury them. The fan-out asks once and never calls

// this for a check.

//

// QUIET BY DEFAULT. Failures and errors are logged, passes are not - eighty green

// lines hide the two that matter, and the counts are already available through

// I_TestRunStatus for anyone who wants them. SetVerbosity(TRUE) if you want the

// narration.

//

// Severity is not decoration. A FAILURE is an error: the code under test was shown

// to be wrong. An ERROR is a warning: the test could not run, so nothing was shown

// about the code at all, and a build should react differently to each.
FUNCTION_BLOCK TestLogReporter IMPLEMENTS I_TestReporter
VAR
	_Prefix				   : T_MaxString;
	_IncludePasses		   : BOOL;
	_LinesWritten		   : UDINT;
	_FailuresLogged		   : UDINT;
	_ErrorsLogged		   : UDINT;
	_FrameworkErrorsLogged : UDINT;

	// The banner rule. Held once so both ends of a run are drawn identically - two

	// rules that differed by a character would be worse than none.
	_Rule		: T_MaxString := '========================================================';
	_TestsSeen	: UDINT;
	_SuitesSeen : UDINT;
END_VAR

(*
	No cyclic body. Everything this sink does happens inside the notification that
	prompted it.
*)

// Nothing to advance. ADSLOGSTR completes within the call, which is what makes

// this the cheapest sink to attach and the safest one to attach first.
METHOD CyclicLogic
(*
	Deliberately empty. This sink starts no asynchronous work, so it has none to
	finish - which is also why IsIdle is always TRUE.
*)
END_METHOD

// The one place anything is written. Private, so severity and destination are

// chosen here and cannot drift between call sites.
METHOD Emit
VAR_INPUT
	Severity : DWORD;
	Line	 : T_MaxString;
END_VAR
// A severity bit alone does not say where the message goes. LOG is what puts it

